    |   movel([0.079939, -1.343105, -2.596200, -0.773084, 1.570796, 1.650735],accel_mss,speed_ms,0,blend_radius_m)
    |   movel([0.079516, -1.343110, -2.596196, -0.773082, 1.570796, 1.650312],accel_mss,speed_ms,0,blend_radius_m)
    |   movel([0.079131, -1.343095, -2.596206, -0.773088, 1.570796, 1.649927],accel_mss,speed_ms,0,blend_radius_m)
    |   movel([0.078857, -1.343061, -2.596229, -0.773099, 1.570796, 1.649653],accel_mss,speed_ms,0,blend_radius_m)
    |   movel([0.077911, -1.342715, -2.596455, -0.773220, 1.570796, 1.648707],accel_mss,speed_ms,0,blend_radius_m)
    |   movel([0.077138, -1.342102, -2.596854, -0.773432, 1.570796, 1.647934],accel_mss,speed_ms,0,blend_radius_m)
    |   movel([0.076602, -1.341277, -2.597392, -0.773720, 1.570796, 1.647398],accel_mss,speed_ms,0,blend_radius_m)
    |   movel([0.076353, -1.340309, -2.598021, -0.774059, 1.570796, 1.647149],accel_mss,speed_ms,0,blend_radius_m)
    |   movel([0.076437, -1.339121, -2.598792, -0.774476, 1.570796, 1.647234],accel_mss,speed_ms,0,blend_radius_m)
    |   movel([0.076894, -1.337754, -2.599676, -0.774958, 1.570796, 1.647690],accel_mss,speed_ms,0,blend_radius_m)
    |   movel([0.077674, -1.336337, -2.600591, -0.775461, 1.570796, 1.648470],accel_mss,speed_ms,0,blend_radius_m)
    |   movel([0.078708, -1.335004, -2.601448, -0.775937, 1.570796, 1.649504],accel_mss,speed_ms,0,blend_radius_m)
    |   movel([0.080811, -1.333153, -2.602635, -0.776601, 1.570796, 1.651607],accel_mss,speed_ms,0,blend_radius_m)
    |   movel([0.083274, -1.331799, -2.603500, -0.777090, 1.570796, 1.654070],accel_mss,speed_ms,0,blend_radius_m)
    |   movel([0.085841, -1.331090, -2.603952, -0.777347, 1.570796, 1.656638],accel_mss,speed_ms,0,blend_radius_m)
    |   movel([0.088231, -1.331107, -2.603941, -0.777341, 1.570796, 1.659028],accel_mss,speed_ms,0,blend_radius_m)
    |   movel([0.089974, -1.331777, -2.603514, -0.777098, 1.570796, 1.660770],accel_mss,speed_ms,0,blend_radius_m)
    |   movel([0.091117, -1.333045, -2.602704, -0.776640, 1.570796, 1.661913],accel_mss,speed_ms,0,blend_radius_m)
    |   movel([0.091521, -1.334728, -2.601626, -0.776036, 1.570796, 1.662317],accel_mss,speed_ms,0,blend_radius_m)
    |   movel([0.091134, -1.336614, -2.600412, -0.775363, 1.570796, 1.661931],accel_mss,speed_ms,0,blend_radius_m)
    |   movel([0.090360, -1.338022, -2.599503, -0.774864, 1.570796, 1.661156],accel_mss,speed_ms,0,blend_radius_m)
    |   movel([0.089237, -1.339332, -2.598656, -0.774402, 1.570796, 1.660033],accel_mss,speed_ms,0,blend_radius_m)
    |   movel([0.087880, -1.340411, -2.597955, -0.774023, 1.570796, 1.658676],accel_mss,speed_ms,0,blend_radius_m)
    |   movel([0.086419, -1.341159, -2.597469, -0.773761, 1.570796, 1.657215],accel_mss,speed_ms,0,blend_radius_m)
    |   movel([0.086085, -1.341294, -2.597381, -0.773714, 1.570796, 1.656881],accel_mss,speed_ms,0,blend_radius_m)
    |   movel([0.085784, -1.341434, -2.597289, -0.773665, 1.570796, 1.656580],accel_mss,speed_ms,0,blend_radius_m)
    |   movel([0.085437, -1.341649, -2.597150, -0.773590, 1.570796, 1.656234],accel_mss,speed_ms,0,blend_radius_m)
    |   movel([0.085272, -1.342062, -2.596880, -0.773446, 1.570796, 1.656068],accel_mss,speed_ms,0,blend_radius_m)
    |   movel([0.085168, -1.342424, -2.596644, -0.773321, 1.570796, 1.655964],accel_mss,speed_ms,0,blend_radius_m)
    |   movel([0.085068, -1.342821, -2.596385, -0.773183, 1.570796, 1.655864],accel_mss,speed_ms,0,blend_radius_m)
    |   movel([0.084872, -1.343546, -2.595911, -0.772931, 1.570796, 1.655669],accel_mss,speed_ms,0,blend_radius_m)
    |   movel([0.084670, -1.343986, -2.595624, -0.772779, 1.570796, 1.655466],accel_mss,speed_ms,0,blend_radius_m)
    |   movel([0.084233, -1.344177, -2.595498, -0.772713, 1.570796, 1.655029],accel_mss,speed_ms,0,blend_radius_m)
    |   movel([0.084159, -1.343630, -2.595857, -0.772903, 1.570796, 1.654955],accel_mss,speed_ms,0,blend_radius_m)
    |   movel([0.084254, -1.342914, -2.596324, -0.773150, 1.570796, 1.655050],accel_mss,speed_ms,0,blend_radius_m)
    |   movel([0.084514, -1.341336, -2.597354, -0.773700, 1.570796, 1.655311],accel_mss,speed_ms,0,blend_radius_m)
    |   movel([0.084702, -1.340274, -2.598044, -0.774071, 1.570796, 1.655498],accel_mss,speed_ms,0,blend_radius_m)
    |   movel([0.084875, -1.339360, -2.598637, -0.774392, 1.570796, 1.655672],accel_mss,speed_ms,0,blend_radius_m)
    |   movel([0.085040, -1.338563, -2.599153, -0.774672, 1.570796, 1.655836],accel_mss,speed_ms,0,blend_radius_m)
    |   movel([0.085311, -1.338276, -2.599339, -0.774774, 1.570796, 1.656107],accel_mss,speed_ms,0,blend_radius_m)
    |   movel([0.085672, -1.338005, -2.599514, -0.774869, 1.570796, 1.656468],accel_mss,speed_ms,0,blend_radius_m)
    |   movel([0.086068, -1.337661, -2.599737, -0.774991, 1.570796, 1.656864],accel_mss,speed_ms,0,blend_radius_m)
    |   movel([0.086444, -1.337219, -2.600022, -0.775148, 1.570796, 1.657240],accel_mss,speed_ms,0,blend_radius_m)
    |   movel([0.086729, -1.336771, -2.600311, -0.775307, 1.570796, 1.657525],accel_mss,speed_ms,0,blend_radius_m)
    |   movel([0.086840, -1.336424, -2.600534, -0.775430, 1.570796, 1.657636],accel_mss,speed_ms,0,blend_radius_m)
    |   movel([0.086756, -1.336163, -2.600703, -0.775523, 1.570796, 1.657553],accel_mss,speed_ms,0,blend_radius_m)
    |   movel([0.086516, -1.335929, -2.600853, -0.775606, 1.570796, 1.657313],accel_mss,speed_ms,0,blend_radius_m)
    |   movel([0.085950, -1.335813, -2.600928, -0.775648, 1.570796, 1.656746],accel_mss,speed_ms,0,blend_radius_m)
    |   movel([0.085372, -1.336061, -2.600768, -0.775559, 1.570796, 1.656169],accel_mss,speed_ms,0,blend_radius_m)
    |   movel([0.084915, -1.336633, -2.600400, -0.775356, 1.570796, 1.655711],accel_mss,speed_ms,0,blend_radius_m)
    |   movel([0.084701, -1.337386, -2.599914, -0.775089, 1.570796, 1.655497],accel_mss,speed_ms,0,blend_radius_m)
    |   movel([0.084629, -1.337702, -2.599710, -0.774977, 1.570796, 1.655425],accel_mss,speed_ms,0,blend_radius_m)
    |   movel([0.084484, -1.338005, -2.599514, -0.774870, 1.570796, 1.655281],accel_mss,speed_ms,0,blend_radius_m)
    |   movel([0.084293, -1.338243, -2.599361, -0.774785, 1.570796, 1.655089],accel_mss,speed_ms,0,blend_radius_m)
    |   movel([0.083838, -1.338404, -2.599256, -0.774729, 1.570796, 1.654634],accel_mss,speed_ms,0,blend_radius_m)
    |   speed_ms = 0.003
    |   movel([0.083838, -1.341807, -2.600812, -0.769770, 1.570796, 1.654634],accel_mss,speed_ms,0,blend_radius_m)
    |   speed_ms = 0.007
    |   movel([0.083575, -1.341756, -2.600845, -0.769788, 1.570796, 1.654371],accel_mss,speed_ms,0,blend_radius_m)
    |   movel([0.083364, -1.341641, -2.600920, -0.769828, 1.570796, 1.654160],accel_mss,speed_ms,0,blend_radius_m)
    |   movel([0.083137, -1.341072, -2.601289, -0.770028, 1.570796, 1.653934],accel_mss,speed_ms,0,blend_radius_m)
    |   movel([0.082925, -1.340755, -2.601495, -0.770139, 1.570796, 1.653721],accel_mss,speed_ms,0,blend_radius_m)
    |   movel([0.082638, -1.340551, -2.601627, -0.770210, 1.570796, 1.653434],accel_mss,speed_ms,0,blend_radius_m)
    |   movel([0.082291, -1.340461, -2.601686, -0.770242, 1.570796, 1.653087],accel_mss,speed_ms,0,blend_radius_m)
    |   movel([0.081838, -1.340482, -2.601672, -0.770235, 1.570796, 1.652635],accel_mss,speed_ms,0,blend_radius_m)
    |   movel([0.081455, -1.340581, -2.601608, -0.770200, 1.570796, 1.652252],accel_mss,speed_ms,0,blend_radius_m)
    |   movel([0.081141, -1.340794, -2.601470, -0.770125, 1.570796, 1.651937],accel_mss,speed_ms,0,blend_radius_m)
    |   movel([0.080784, -1.341164, -2.601229, -0.769995, 1.570796, 1.651580],accel_mss,speed_ms,0,blend_radius_m)
    |   movel([0.080489, -1.341559, -2.600973, -0.769857, 1.570796, 1.651285],accel_mss,speed_ms,0,blend_radius_m)
    |   movel([0.080384, -1.341838, -2.600791, -0.769759, 1.570796, 1.651180],accel_mss,speed_ms,0,blend_radius_m)
    |   movel([0.080469, -1.342126, -2.600605, -0.769659, 1.570796, 1.651266],accel_mss,speed_ms,0,blend_radius_m)
    |   movel([0.080802, -1.342368, -2.600447, -0.769574, 1.570796, 1.651598],accel_mss,speed_ms,0,blend_radius_m)
    |   movel([0.081280, -1.342524, -2.600345, -0.769520, 1.570796, 1.652076],accel_mss,speed_ms,0,blend_radius_m)
    |   movel([0.081829, -1.342556, -2.600324, -0.769508, 1.570796, 1.652625],accel_mss,speed_ms,0,blend_radius_m)
    |   movel([0.082528, -1.342582, -2.600308, -0.769500, 1.570796, 1.653324],accel_mss,speed_ms,0,blend_radius_m)
    |   movel([0.082794, -1.342792, -2.600170, -0.769426, 1.570796, 1.653590],accel_mss,speed_ms,0,blend_radius_m)
    |   movel([0.082846, -1.343313, -2.599831, -0.769245, 1.570796, 1.653642],accel_mss,speed_ms,0,blend_radius_m)
    |   movel([0.082677, -1.345239, -2.598572, -0.768578, 1.570796, 1.653473],accel_mss,speed_ms,0,blend_radius_m)
    |   movel([0.082499, -1.346941, -2.597455, -0.767993, 1.570796, 1.653295],accel_mss,speed_ms,0,blend_radius_m)
    |   movel([0.082356, -1.347693, -2.596960, -0.767736, 1.570796, 1.653152],accel_mss,speed_ms,0,blend_radius_m)
    |   movel([0.082163, -1.348091, -2.596698, -0.767600, 1.570796, 1.652960],accel_mss,speed_ms,0,blend_radius_m)
    |   movel([0.081866, -1.348309, -2.596554, -0.767525, 1.570796, 1.652662],accel_mss,speed_ms,0,blend_radius_m)
    |   movel([0.081568, -1.348137, -2.596668, -0.767584, 1.570796, 1.652364],accel_mss,speed_ms,0,blend_radius_m)
    |   movel([0.081509, -1.347824, -2.596874, -0.767691, 1.570796, 1.652305],accel_mss,speed_ms,0,blend_radius_m)
    |   movel([0.081511, -1.347338, -2.597194, -0.767857, 1.570796, 1.652308],accel_mss,speed_ms,0,blend_radius_m)
    |   movel([0.081515, -1.347062, -2.597375, -0.767951, 1.570796, 1.652311],accel_mss,speed_ms,0,blend_radius_m)
    |   movel([0.081498, -1.346808, -2.597542, -0.768038, 1.570796, 1.652294],accel_mss,speed_ms,0,blend_radius_m)
    |   movel([0.081461, -1.346604, -2.597676, -0.768108, 1.570796, 1.652258],accel_mss,speed_ms,0,blend_radius_m)
    |   movel([0.081307, -1.346463, -2.597769, -0.768157, 1.570796, 1.652103],accel_mss,speed_ms,0,blend_radius_m)
    |   movel([0.081039, -1.346444, -2.597782, -0.768163, 1.570796, 1.651836],accel_mss,speed_ms,0,blend_radius_m)
    |   movel([0.080706, -1.346443, -2.597782, -0.768164, 1.570796, 1.651503],accel_mss,speed_ms,0,blend_radius_m)
    |   movel([0.080338, -1.346469, -2.597765, -0.768155, 1.570796, 1.651134],accel_mss,speed_ms,0,blend_radius_m)
    |   movel([0.079939, -1.346496, -2.597748, -0.768146, 1.570796, 1.650735],accel_mss,speed_ms,0,blend_radius_m)
    |   movel([0.079516, -1.346501, -2.597744, -0.768144, 1.570796, 1.650312],accel_mss,speed_ms,0,blend_radius_m)
    |   movel([0.079131, -1.346486, -2.597754, -0.768149, 1.570796, 1.649927],accel_mss,speed_ms,0,blend_radius_m)
    |   movel([0.078857, -1.346452, -2.597776, -0.768161, 1.570796, 1.649653],accel_mss,speed_ms,0,blend_radius_m)
    |   movel([0.077911, -1.346107, -2.598003, -0.768279, 1.570796, 1.648707],accel_mss,speed_ms,0,blend_radius_m)
    |   movel([0.077138, -1.345496, -2.598404, -0.768490, 1.570796, 1.647934],accel_mss,speed_ms,0,blend_radius_m)
    |   movel([0.076602, -1.344673, -2.598942, -0.768774, 1.570796, 1.647398],accel_mss,speed_ms,0,blend_radius_m)
    |   movel([0.076353, -1.343707, -2.599574, -0.769108, 1.570796, 1.647149],accel_mss,speed_ms,0,blend_radius_m)
    |   movel([0.076437, -1.342522, -2.600346, -0.769520, 1.570796, 1.647234],accel_mss,speed_ms,0,blend_radius_m)
    |   movel([0.076894, -1.341159, -2.601233, -0.769997, 1.570796, 1.647690],accel_mss,speed_ms,0,blend_radius_m)
    |   movel([0.077674, -1.339745, -2.602150, -0.770494, 1.570796, 1.648470],accel_mss,speed_ms,0,blend_radius_m)
    |   movel([0.078708, -1.338415, -2.603009, -0.770964, 1.570796, 1.649504],accel_mss,speed_ms,0,blend_radius_m)
    |   movel([0.080811, -1.336569, -2.604199, -0.771621, 1.570796, 1.651607],accel_mss,speed_ms,0,blend_radius_m)
    |   movel([0.083274, -1.335218, -2.605067, -0.772104, 1.570796, 1.654070],accel_mss,speed_ms,0,blend_radius_m)
    |   movel([0.085841, -1.334511, -2.605520, -0.772358, 1.570796, 1.656638],accel_mss,speed_ms,0,blend_radius_m)
    |   movel([0.088231, -1.334527, -2.605509, -0.772352, 1.570796, 1.659028],accel_mss,speed_ms,0,blend_radius_m)
    |   movel([0.089974, -1.335197, -2.605081, -0.772112, 1.570796, 1.660770],accel_mss,speed_ms,0,blend_radius_m)
    |   movel([0.091117, -1.336461, -2.604269, -0.771659, 1.570796, 1.661913],accel_mss,speed_ms,0,blend_radius_m)
    |   movel([0.091521, -1.338140, -2.603187, -0.771062, 1.570796, 1.662317],accel_mss,speed_ms,0,blend_radius_m)
    |   movel([0.091134, -1.340021, -2.601971, -0.770397, 1.570796, 1.661931],accel_mss,speed_ms,0,blend_radius_m)
    |   movel([0.090360, -1.341426, -2.601060, -0.769904, 1.570796, 1.661156],accel_mss,speed_ms,0,blend_radius_m)
    |   movel([0.089237, -1.342732, -2.600210, -0.769447, 1.570796, 1.660033],accel_mss,speed_ms,0,blend_radius_m)
    |   movel([0.087880, -1.343808, -2.599508, -0.769073, 1.570796, 1.658676],accel_mss,speed_ms,0,blend_radius_m)
    |   movel([0.086419, -1.344555, -2.599020, -0.768814, 1.570796, 1.657215],accel_mss,speed_ms,0,blend_radius_m)
    |   movel([0.086085, -1.344690, -2.598932, -0.768768, 1.570796, 1.656881],accel_mss,speed_ms,0,blend_radius_m)
    |   movel([0.085784, -1.344830, -2.598840, -0.768719, 1.570796, 1.656580],accel_mss,speed_ms,0,blend_radius_m)
    |   movel([0.085437, -1.345043, -2.598700, -0.768646, 1.570796, 1.656234],accel_mss,speed_ms,0,blend_radius_m)
    |   movel([0.085272, -1.345456, -2.598430, -0.768503, 1.570796, 1.656068],accel_mss,speed_ms,0,blend_radius_m)
    |   movel([0.085168, -1.345817, -2.598193, -0.768379, 1.570796, 1.655964],accel_mss,speed_ms,0,blend_radius_m)
    |   movel([0.085068, -1.346213, -2.597933, -0.768243, 1.570796, 1.655864],accel_mss,speed_ms,0,blend_radius_m)
    |   movel([0.084872, -1.346936, -2.597458, -0.767995, 1.570796, 1.655669],accel_mss,speed_ms,0,blend_radius_m)
    |   movel([0.084670, -1.347375, -2.597170, -0.767844, 1.570796, 1.655466],accel_mss,speed_ms,0,blend_radius_m)
    |   movel([0.084233, -1.347565, -2.597044, -0.767779, 1.570796, 1.655029],accel_mss,speed_ms,0,blend_radius_m)
    |   movel([0.084159, -1.347019, -2.597404, -0.767966, 1.570796, 1.654955],accel_mss,speed_ms,0,blend_radius_m)
    |   movel([0.084254, -1.346306, -2.597872, -0.768211, 1.570796, 1.655050],accel_mss,speed_ms,0,blend_radius_m)
    |   movel([0.084514, -1.344731, -2.598904, -0.768754, 1.570796, 1.655311],accel_mss,speed_ms,0,blend_radius_m)
    |   movel([0.084702, -1.343673, -2.599596, -0.769120, 1.570796, 1.655498],accel_mss,speed_ms,0,blend_radius_m)
    |   movel([0.084875, -1.342761, -2.600191, -0.769437, 1.570796, 1.655672],accel_mss,speed_ms,0,blend_radius_m)
    |   movel([0.085040, -1.341966, -2.600709, -0.769715, 1.570796, 1.655836],accel_mss,speed_ms,0,blend_radius_m)
    |   movel([0.085311, -1.341679, -2.600895, -0.769815, 1.570796, 1.656107],accel_mss,speed_ms,0,blend_radius_m)
    |   movel([0.085672, -1.341409, -2.601070, -0.769909, 1.570796, 1.656468],accel_mss,speed_ms,0,blend_radius_m)
    |   movel([0.086068, -1.341066, -2.601294, -0.770030, 1.570796, 1.656864],accel_mss,speed_ms,0,blend_radius_m)
    |   movel([0.086444, -1.340624, -2.601580, -0.770185, 1.570796, 1.657240],accel_mss,speed_ms,0,blend_radius_m)
    |   movel([0.086729, -1.340178, -2.601869, -0.770342, 1.570796, 1.657525],accel_mss,speed_ms,0,blend_radius_m)
    |   movel([0.086840, -1.339832, -2.602093, -0.770464, 1.570796, 1.657636],accel_mss,speed_ms,0,blend_radius_m)
    |   movel([0.086756, -1.339572, -2.602262, -0.770555, 1.570796, 1.657553],accel_mss,speed_ms,0,blend_radius_m)
    |   movel([0.086516, -1.339338, -2.602413, -0.770638, 1.570796, 1.657313],accel_mss,speed_ms,0,blend_radius_m)
    |   movel([0.085950, -1.339222, -2.602488, -0.770679, 1.570796, 1.656746],accel_mss,speed_ms,0,blend_radius_m)
    |   movel([0.085372, -1.339470, -2.602328, -0.770591, 1.570796, 1.656169],accel_mss,speed_ms,0,blend_radius_m)
    |   movel([0.084915, -1.340040, -2.601959, -0.770390, 1.570796, 1.655711],accel_mss,speed_ms,0,blend_radius_m)
    |   movel([0.084701, -1.340791, -2.601472, -0.770126, 1.570796, 1.655497],accel_mss,speed_ms,0,blend_radius_m)
    |   movel([0.084629, -1.341106, -2.601267, -0.770016, 1.570796, 1.655425],accel_mss,speed_ms,0,blend_radius_m)
    |   movel([0.084484, -1.341409, -2.601071, -0.769910, 1.570796, 1.655281],accel_mss,speed_ms,0,blend_radius_m)
    |   movel([0.084293, -1.341646, -2.600916, -0.769826, 1.570796, 1.655089],accel_mss,speed_ms,0,blend_radius_m)
    |   movel([0.083838, -1.341807, -2.600812, -0.769770, 1.570796, 1.654634],accel_mss,speed_ms,0,blend_radius_m)
    |   speed_ms = 0.003
    |   movel([0.083838, -1.328347, -2.594539, -0.789503, 1.570796, 1.654634],accel_mss,speed_ms,0,blend_radius_m)
    |   speed_ms = 1.000
    |   movel([0.083838, -1.302622, -2.581603, -0.828165, 1.570796, 1.654634],accel_mss,speed_ms,0,blend_radius_m)
    |   movel([0.083131, -1.309400, -2.577409, -0.825580, 1.570796, 1.653928],accel_mss,speed_ms,0,blend_radius_m)
    |   movel([0.083131, -1.335017, -2.590258, -0.787114, 1.570796, 1.653928],accel_mss,speed_ms,0,blend_radius_m)
    |   speed_ms = 0.003
    |   movel([0.083131, -1.345027, -2.594942, -0.772421, 1.570796, 1.653928],accel_mss,speed_ms,0,blend_radius_m)
    |   speed_ms = 0.007
    |   movel([0.084912, -1.344646, -2.595191, -0.772552, 1.570796, 1.655708],accel_mss,speed_ms,0,blend_radius_m)
    |   movel([0.085226, -1.344667, -2.595177, -0.772544, 1.570796, 1.656023],accel_mss,speed_ms,0,blend_radius_m)
    |   movel([0.085321, -1.344944, -2.594996, -0.772449, 1.570796, 1.656117],accel_mss,speed_ms,0,blend_radius_m)
    |   movel([0.085214, -1.345307, -2.594758, -0.772325, 1.570796, 1.656010],accel_mss,speed_ms,0,blend_radius_m)
    |   movel([0.085158, -1.345566, -2.594588, -0.772236, 1.570796, 1.655955],accel_mss,speed_ms,0,blend_radius_m)
    |   movel([0.085106, -1.345844, -2.594405, -0.772140, 1.570796, 1.655902],accel_mss,speed_ms,0,blend_radius_m)
    |   movel([0.085067, -1.346106, -2.594233, -0.772050, 1.570796, 1.655864],accel_mss,speed_ms,0,blend_radius_m)
    |   movel([0.085015, -1.346429, -2.594020, -0.771940, 1.570796, 1.655812],accel_mss,speed_ms,0,blend_radius_m)
    |   movel([0.084839, -1.346835, -2.593753, -0.771801, 1.570796, 1.655635],accel_mss,speed_ms,0,blend_radius_m)
    |   movel([0.084290, -1.347303, -2.593444, -0.771641, 1.570796, 1.655087],accel_mss,speed_ms,0,blend_radius_m)
    |   movel([0.083746, -1.347575, -2.593265, -0.771549, 1.570796, 1.654542],accel_mss,speed_ms,0,blend_radius_m)
    |   movel([0.083025, -1.347847, -2.593086, -0.771456, 1.570796, 1.653821],accel_mss,speed_ms,0,blend_radius_m)
    |   movel([0.082091, -1.348128, -2.592900, -0.771361, 1.570796, 1.652888],accel_mss,speed_ms,0,blend_radius_m)
    |   movel([0.081241, -1.348334, -2.592764, -0.771291, 1.570796, 1.652037],accel_mss,speed_ms,0,blend_radius_m)
    |   movel([0.080813, -1.348339, -2.592761, -0.771289, 1.570796, 1.651610],accel_mss,speed_ms,0,blend_radius_m)
    |   movel([0.080675, -1.348167, -2.592874, -0.771347, 1.570796, 1.651471],accel_mss,speed_ms,0,blend_radius_m)
    |   movel([0.080768, -1.347825, -2.593100, -0.771464, 1.570796, 1.651564],accel_mss,speed_ms,0,blend_radius_m)
    |   movel([0.080890, -1.347520, -2.593302, -0.771568, 1.570796, 1.651686],accel_mss,speed_ms,0,blend_radius_m)
    |   movel([0.080645, -1.347327, -2.593429, -0.771633, 1.570796, 1.651441],accel_mss,speed_ms,0,blend_radius_m)
    |   movel([0.080619, -1.347111, -2.593571, -0.771707, 1.570796, 1.651416],accel_mss,speed_ms,0,blend_radius_m)
    |   movel([0.080919, -1.346779, -2.593790, -0.771820, 1.570796, 1.651715],accel_mss,speed_ms,0,blend_radius_m)
    |   movel([0.080769, -1.346426, -2.594022, -0.771941, 1.570796, 1.651566],accel_mss,speed_ms,0,blend_radius_m)
    |   movel([0.080640, -1.346238, -2.594146, -0.772005, 1.570796, 1.651436],accel_mss,speed_ms,0,blend_radius_m)
    |   movel([0.080628, -1.346014, -2.594293, -0.772082, 1.570796, 1.651424],accel_mss,speed_ms,0,blend_radius_m)
    |   movel([0.080942, -1.345606, -2.594561, -0.772222, 1.570796, 1.651739],accel_mss,speed_ms,0,blend_radius_m)
    |   movel([0.081368, -1.345424, -2.594681, -0.772284, 1.570796, 1.652164],accel_mss,speed_ms,0,blend_radius_m)
    |   movel([0.083131, -1.345027, -2.594942, -0.772421, 1.570796, 1.653928],accel_mss,speed_ms,0,blend_radius_m)
    |   speed_ms = 0.003
    |   movel([0.083131, -1.348413, -2.596486, -0.767490, 1.570796, 1.653928],accel_mss,speed_ms,0,blend_radius_m)
    |   speed_ms = 0.007
    |   movel([0.084912, -1.348033, -2.596736, -0.767620, 1.570796, 1.655708],accel_mss,speed_ms,0,blend_radius_m)
    |   movel([0.085226, -1.348054, -2.596722, -0.767612, 1.570796, 1.656023],accel_mss,speed_ms,0,blend_radius_m)
    |   movel([0.085321, -1.348330, -2.596541, -0.767518, 1.570796, 1.656117],accel_mss,speed_ms,0,blend_radius_m)
    |   movel([0.085214, -1.348692, -2.596302, -0.767395, 1.570796, 1.656010],accel_mss,speed_ms,0,blend_radius_m)
    |   movel([0.085158, -1.348950, -2.596131, -0.767307, 1.570796, 1.655955],accel_mss,speed_ms,0,blend_radius_m)
    |   movel([0.085106, -1.349228, -2.595948, -0.767213, 1.570796, 1.655902],accel_mss,speed_ms,0,blend_radius_m)
    |   movel([0.085067, -1.349489, -2.595775, -0.767124, 1.570796, 1.655864],accel_mss,speed_ms,0,blend_radius_m)
    |   movel([0.085015, -1.349812, -2.595562, -0.767015, 1.570796, 1.655812],accel_mss,speed_ms,0,blend_radius_m)
    |   movel([0.084839, -1.350216, -2.595294, -0.766878, 1.570796, 1.655635],accel_mss,speed_ms,0,blend_radius_m)
    |   movel([0.084290, -1.350683, -2.594985, -0.766720, 1.570796, 1.655087],accel_mss,speed_ms,0,blend_radius_m)
    |   movel([0.083746, -1.350954, -2.594806, -0.766629, 1.570796, 1.654542],accel_mss,speed_ms,0,blend_radius_m)
    |   movel([0.083025, -1.351226, -2.594626, -0.766538, 1.570796, 1.653821],accel_mss,speed_ms,0,blend_radius_m)
    |   movel([0.082091, -1.351507, -2.594439, -0.766443, 1.570796, 1.652888],accel_mss,speed_ms,0,blend_radius_m)
    |   movel([0.081241, -1.351712, -2.594303, -0.766374, 1.570796, 1.652037],accel_mss,speed_ms,0,blend_radius_m)
    |   movel([0.080813, -1.351716, -2.594300, -0.766373, 1.570796, 1.651610],accel_mss,speed_ms,0,blend_radius_m)
    |   movel([0.080675, -1.351545, -2.594414, -0.766430, 1.570796, 1.651471],accel_mss,speed_ms,0,blend_radius_m)
    |   movel([0.080768, -1.351204, -2.594640, -0.766545, 1.570796, 1.651564],accel_mss,speed_ms,0,blend_radius_m)
    |   movel([0.080890, -1.350900, -2.594842, -0.766647, 1.570796, 1.651686],accel_mss,speed_ms,0,blend_radius_m)
    |   movel([0.080645, -1.350707, -2.594969, -0.766712, 1.570796, 1.651441],accel_mss,speed_ms,0,blend_radius_m)
    |   movel([0.080619, -1.350492, -2.595112, -0.766785, 1.570796, 1.651416],accel_mss,speed_ms,0,blend_radius_m)
    |   movel([0.080919, -1.350160, -2.595332, -0.766897, 1.570796, 1.651715],accel_mss,speed_ms,0,blend_radius_m)
    |   movel([0.080769, -1.349809, -2.595564, -0.767016, 1.570796, 1.651566],accel_mss,speed_ms,0,blend_radius_m)
    |   movel([0.080640, -1.349621, -2.595688, -0.767080, 1.570796, 1.651436],accel_mss,speed_ms,0,blend_radius_m)
    |   movel([0.080628, -1.349397, -2.595836, -0.767155, 1.570796, 1.651424],accel_mss,speed_ms,0,blend_radius_m)
    |   movel([0.080942, -1.348990, -2.596105, -0.767294, 1.570796, 1.651739],accel_mss,speed_ms,0,blend_radius_m)
    |   movel([0.081368, -1.348809, -2.596225, -0.767355, 1.570796, 1.652164],accel_mss,speed_ms,0,blend_radius_m)
    |   movel([0.083131, -1.348413, -2.596486, -0.767490, 1.570796, 1.653928],accel_mss,speed_ms,0,blend_radius_m)
    |   speed_ms = 0.003
    |   movel([0.083131, -1.335017, -2.590258, -0.787114, 1.570796, 1.653928],accel_mss,speed_ms,0,blend_radius_m)
    |   speed_ms = 1.000
    |   movel([0.083131, -1.309400, -2.577409, -0.825580, 1.570796, 1.653928],accel_mss,speed_ms,0,blend_radius_m)
    |   movel([0.082638, -1.312886, -2.575230, -0.824273, 1.570796, 1.653435],accel_mss,speed_ms,0,blend_radius_m)
    |   movel([0.082638, -1.338446, -2.588033, -0.785910, 1.570796, 1.653435],accel_mss,speed_ms,0,blend_radius_m)
    |   speed_ms = 0.003
    |   movel([0.082638, -1.348431, -2.592700, -0.771258, 1.570796, 1.653435],accel_mss,speed_ms,0,blend_radius_m)
    |   speed_ms = 0.007
    |   movel([0.083010, -1.348325, -2.592770, -0.771294, 1.570796, 1.653806],accel_mss,speed_ms,0,blend_radius_m)
    |   movel([0.083255, -1.348397, -2.592722, -0.771269, 1.570796, 1.654051],accel_mss,speed_ms,0,blend_radius_m)
    |   movel([0.083272, -1.348613, -2.592580, -0.771196, 1.570796, 1.654068],accel_mss,speed_ms,0,blend_radius_m)
    |   movel([0.082991, -1.348882, -2.592402, -0.771105, 1.570796, 1.653788],accel_mss,speed_ms,0,blend_radius_m)
    |   movel([0.082561, -1.349059, -2.592285, -0.771045, 1.570796, 1.653357],accel_mss,speed_ms,0,blend_radius_m)
    |   movel([0.082329, -1.349028, -2.592305, -0.771056, 1.570796, 1.653125],accel_mss,speed_ms,0,blend_radius_m)
    |   movel([0.082337, -1.348676, -2.592538, -0.771175, 1.570796, 1.653134],accel_mss,speed_ms,0,blend_radius_m)
    |   movel([0.082638, -1.348431, -2.592700, -0.771258, 1.570796, 1.653435],accel_mss,speed_ms,0,blend_radius_m)
    |   speed_ms = 0.003
    |   movel([0.082638, -1.351808, -2.594239, -0.766342, 1.570796, 1.653435],accel_mss,speed_ms,0,blend_radius_m)
    |   speed_ms = 0.007
    |   movel([0.083010, -1.351702, -2.594309, -0.766377, 1.570796, 1.653806],accel_mss,speed_ms,0,blend_radius_m)
    |   movel([0.083255, -1.351775, -2.594261, -0.766353, 1.570796, 1.654051],accel_mss,speed_ms,0,blend_radius_m)
    |   movel([0.083272, -1.351990, -2.594118, -0.766281, 1.570796, 1.654068],accel_mss,speed_ms,0,blend_radius_m)
    |   movel([0.082991, -1.352258, -2.593940, -0.766191, 1.570796, 1.653788],accel_mss,speed_ms,0,blend_radius_m)
    |   movel([0.082561, -1.352435, -2.593823, -0.766132, 1.570796, 1.653357],accel_mss,speed_ms,0,blend_radius_m)
    |   movel([0.082329, -1.352404, -2.593843, -0.766142, 1.570796, 1.653125],accel_mss,speed_ms,0,blend_radius_m)
    |   movel([0.082337, -1.352052, -2.594077, -0.766260, 1.570796, 1.653134],accel_mss,speed_ms,0,blend_radius_m)
    |   movel([0.082638, -1.351808, -2.594239, -0.766342, 1.570796, 1.653435],accel_mss,speed_ms,0,blend_radius_m)
    |   speed_ms = 0.003
    |   movel([0.082638, -1.338446, -2.588033, -0.785910, 1.570796, 1.653435],accel_mss,speed_ms,0,blend_radius_m)
    |   speed_ms = 1.000
    |   movel([0.082638, -1.312886, -2.575230, -0.824273, 1.570796, 1.653435],accel_mss,speed_ms,0,blend_radius_m)
    |   movel([0.075847, -1.319560, -2.571014, -0.821815, 1.570796, 1.646643],accel_mss,speed_ms,0,blend_radius_m)
    |   movel([0.075847, -1.345010, -2.583731, -0.783648, 1.570796, 1.646643],accel_mss,speed_ms,0,blend_radius_m)
    |   speed_ms = 0.003
    |   movel([0.075847, -1.354947, -2.588365, -0.769077, 1.570796, 1.646643],accel_mss,speed_ms,0,blend_radius_m)
    |   speed_ms = 0.007
    |   movel([0.076210, -1.355243, -2.588167, -0.768979, 1.570796, 1.647006],accel_mss,speed_ms,0,blend_radius_m)
    |   movel([0.076357, -1.355481, -2.588008, -0.768901, 1.570796, 1.647154],accel_mss,speed_ms,0,blend_radius_m)
    |   movel([0.076398, -1.355704, -2.587858, -0.768827, 1.570796, 1.647194],accel_mss,speed_ms,0,blend_radius_m)
    |   movel([0.076337, -1.355959, -2.587687, -0.768743, 1.570796, 1.647134],accel_mss,speed_ms,0,blend_radius_m)
    |   movel([0.076172, -1.356294, -2.587462, -0.768633, 1.570796, 1.646969],accel_mss,speed_ms,0,blend_radius_m)
    |   movel([0.075752, -1.356855, -2.587085, -0.768449, 1.570796, 1.646548],accel_mss,speed_ms,0,blend_radius_m)
    |   movel([0.075239, -1.357270, -2.586806, -0.768313, 1.570796, 1.646035],accel_mss,speed_ms,0,blend_radius_m)
    |   movel([0.074675, -1.357502, -2.586649, -0.768238, 1.570796, 1.645471],accel_mss,speed_ms,0,blend_radius_m)
    |   movel([0.074114, -1.357533, -2.586628, -0.768227, 1.570796, 1.644910],accel_mss,speed_ms,0,blend_radius_m)
    |   movel([0.073609, -1.357253, -2.586817, -0.768319, 1.570796, 1.644405],accel_mss,speed_ms,0,blend_radius_m)
    |   movel([0.073464, -1.356659, -2.587216, -0.768513, 1.570796, 1.644260],accel_mss,speed_ms,0,blend_radius_m)
    |   movel([0.073721, -1.355938, -2.587701, -0.768750, 1.570796, 1.644518],accel_mss,speed_ms,0,blend_radius_m)
    |   movel([0.074305, -1.355315, -2.588118, -0.768955, 1.570796, 1.645101],accel_mss,speed_ms,0,blend_radius_m)
    |   movel([0.074876, -1.354985, -2.588340, -0.769064, 1.570796, 1.645673],accel_mss,speed_ms,0,blend_radius_m)
    |   movel([0.075398, -1.354858, -2.588425, -0.769106, 1.570796, 1.646194],accel_mss,speed_ms,0,blend_radius_m)
    |   movel([0.075847, -1.354947, -2.588365, -0.769077, 1.570796, 1.646643],accel_mss,speed_ms,0,blend_radius_m)
    |   speed_ms = 0.003
    |   movel([0.075847, -1.358308, -2.589893, -0.764188, 1.570796, 1.646643],accel_mss,speed_ms,0,blend_radius_m)
    |   speed_ms = 0.007
    |   movel([0.076210, -1.358603, -2.589694, -0.764092, 1.570796, 1.647006],accel_mss,speed_ms,0,blend_radius_m)
    |   movel([0.076357, -1.358840, -2.589535, -0.764014, 1.570796, 1.647154],accel_mss,speed_ms,0,blend_radius_m)
    |   movel([0.076398, -1.359063, -2.589385, -0.763942, 1.570796, 1.647194],accel_mss,speed_ms,0,blend_radius_m)
    |   movel([0.076337, -1.359317, -2.589213, -0.763859, 1.570796, 1.647134],accel_mss,speed_ms,0,blend_radius_m)
    |   movel([0.076172, -1.359651, -2.588988, -0.763751, 1.570796, 1.646969],accel_mss,speed_ms,0,blend_radius_m)
    |   movel([0.075752, -1.360211, -2.588610, -0.763569, 1.570796, 1.646548],accel_mss,speed_ms,0,blend_radius_m)
    |   movel([0.075239, -1.360624, -2.588330, -0.763435, 1.570796, 1.646035],accel_mss,speed_ms,0,blend_radius_m)
    |   movel([0.074675, -1.360856, -2.588173, -0.763360, 1.570796, 1.645471],accel_mss,speed_ms,0,blend_radius_m)
    |   movel([0.074114, -1.360887, -2.588152, -0.763350, 1.570796, 1.644910],accel_mss,speed_ms,0,blend_radius_m)
    |   movel([0.073609, -1.360608, -2.588341, -0.763440, 1.570796, 1.644405],accel_mss,speed_ms,0,blend_radius_m)
    |   movel([0.073464, -1.360015, -2.588742, -0.763632, 1.570796, 1.644260],accel_mss,speed_ms,0,blend_radius_m)
    |   movel([0.073721, -1.359296, -2.589227, -0.763866, 1.570796, 1.644518],accel_mss,speed_ms,0,blend_radius_m)
    |   movel([0.074305, -1.358675, -2.589646, -0.764068, 1.570796, 1.645101],accel_mss,speed_ms,0,blend_radius_m)
    |   movel([0.074876, -1.358345, -2.589868, -0.764176, 1.570796, 1.645673],accel_mss,speed_ms,0,blend_radius_m)
    |   movel([0.075398, -1.358219, -2.589953, -0.764217, 1.570796, 1.646194],accel_mss,speed_ms,0,blend_radius_m)
    |   movel([0.075847, -1.358308, -2.589893, -0.764188, 1.570796, 1.646643],accel_mss,speed_ms,0,blend_radius_m)
    |   speed_ms = 0.003
    |   movel([0.075847, -1.345010, -2.583731, -0.783648, 1.570796, 1.646643],accel_mss,speed_ms,0,blend_radius_m)
    |   speed_ms = 1.000
    |   movel([0.075847, -1.319560, -2.571014, -0.821815, 1.570796, 1.646643],accel_mss,speed_ms,0,blend_radius_m)
    |   movel([0.078635, -1.323961, -2.568202, -0.820226, 1.570796, 1.649431],accel_mss,speed_ms,0,blend_radius_m)
    |   movel([0.078635, -1.349337, -2.580862, -0.782189, 1.570796, 1.649431],accel_mss,speed_ms,0,blend_radius_m)
    |   speed_ms = 0.003
    |   movel([0.078635, -1.359242, -2.585475, -0.767671, 1.570796, 1.649431],accel_mss,speed_ms,0,blend_radius_m)
    |   speed_ms = 0.007
    |   movel([0.079474, -1.359723, -2.585151, -0.767516, 1.570796, 1.650271],accel_mss,speed_ms,0,blend_radius_m)
    |   movel([0.080172, -1.360238, -2.584802, -0.767349, 1.570796, 1.650969],accel_mss,speed_ms,0,blend_radius_m)
    |   movel([0.080222, -1.360455, -2.584655, -0.767279, 1.570796, 1.651018],accel_mss,speed_ms,0,blend_radius_m)
    |   movel([0.079954, -1.360655, -2.584519, -0.767215, 1.570796, 1.650750],accel_mss,speed_ms,0,blend_radius_m)
    |   movel([0.079275, -1.360021, -2.584949, -0.767419, 1.570796, 1.650071],accel_mss,speed_ms,0,blend_radius_m)
    |   movel([0.078610, -1.359377, -2.585384, -0.767628, 1.570796, 1.649406],accel_mss,speed_ms,0,blend_radius_m)
    |   speed_ms = 0.003
    |   movel([0.078635, -1.362592, -2.586996, -0.762801, 1.570796, 1.649431],accel_mss,speed_ms,0,blend_radius_m)
    |   speed_ms = 0.007
    |   movel([0.079474, -1.363071, -2.586671, -0.762648, 1.570796, 1.650271],accel_mss,speed_ms,0,blend_radius_m)
    |   movel([0.080172, -1.363585, -2.586321, -0.762483, 1.570796, 1.650969],accel_mss,speed_ms,0,blend_radius_m)
    |   movel([0.080222, -1.363801, -2.586174, -0.762414, 1.570796, 1.651018],accel_mss,speed_ms,0,blend_radius_m)
    |   movel([0.079954, -1.364001, -2.586038, -0.762350, 1.570796, 1.650750],accel_mss,speed_ms,0,blend_radius_m)
    |   movel([0.079275, -1.363368, -2.586468, -0.762552, 1.570796, 1.650071],accel_mss,speed_ms,0,blend_radius_m)
    |   movel([0.078610, -1.362726, -2.586905, -0.762758, 1.570796, 1.649406],accel_mss,speed_ms,0,blend_radius_m)
    |   speed_ms = 0.003
    |   movel([0.078635, -1.349337, -2.580862, -0.782189, 1.570796, 1.649431],accel_mss,speed_ms,0,blend_radius_m)
    |   speed_ms = 1.000
    |   movel([0.078635, -1.323961, -2.568202, -0.820226, 1.570796, 1.649431],accel_mss,speed_ms,0,blend_radius_m)
    |   movel([0.084889, -1.331749, -2.563164, -0.817476, 1.570796, 1.655685],accel_mss,speed_ms,0,blend_radius_m)
    |   movel([0.084889, -1.356993, -2.575725, -0.779672, 1.570796, 1.655685],accel_mss,speed_ms,0,blend_radius_m)
    |   speed_ms = 0.003
    |   movel([0.084889, -1.366841, -2.580300, -0.765248, 1.570796, 1.655685],accel_mss,speed_ms,0,blend_radius_m)
    |   speed_ms = 0.007
    |   movel([0.085264, -1.366718, -2.580384, -0.765287, 1.570796, 1.656061],accel_mss,speed_ms,0,blend_radius_m)
    |   movel([0.085429, -1.367001, -2.580190, -0.765198, 1.570796, 1.656225],accel_mss,speed_ms,0,blend_radius_m)
    |   movel([0.085290, -1.367254, -2.580016, -0.765119, 1.570796, 1.656086],accel_mss,speed_ms,0,blend_radius_m)
    |   movel([0.085006, -1.367407, -2.579911, -0.765071, 1.570796, 1.655802],accel_mss,speed_ms,0,blend_radius_m)
    |   movel([0.084700, -1.367358, -2.579945, -0.765087, 1.570796, 1.655496],accel_mss,speed_ms,0,blend_radius_m)
    |   movel([0.084687, -1.367140, -2.580094, -0.765155, 1.570796, 1.655483],accel_mss,speed_ms,0,blend_radius_m)
    |   movel([0.084889, -1.366841, -2.580300, -0.765248, 1.570796, 1.655685],accel_mss,speed_ms,0,blend_radius_m)
    |   speed_ms = 0.003
    |   movel([0.084889, -1.370170, -2.581808, -0.760411, 1.570796, 1.655685],accel_mss,speed_ms,0,blend_radius_m)
    |   speed_ms = 0.007
    |   movel([0.085264, -1.370048, -2.581893, -0.760449, 1.570796, 1.656061],accel_mss,speed_ms,0,blend_radius_m)
    |   movel([0.085429, -1.370330, -2.581698, -0.760361, 1.570796, 1.656225],accel_mss,speed_ms,0,blend_radius_m)
    |   movel([0.085290, -1.370582, -2.581524, -0.760283, 1.570796, 1.656086],accel_mss,speed_ms,0,blend_radius_m)
    |   movel([0.085006, -1.370735, -2.581418, -0.760236, 1.570796, 1.655802],accel_mss,speed_ms,0,blend_radius_m)
    |   movel([0.084700, -1.370686, -2.581452, -0.760251, 1.570796, 1.655496],accel_mss,speed_ms,0,blend_radius_m)
    |   movel([0.084687, -1.370469, -2.581602, -0.760318, 1.570796, 1.655483],accel_mss,speed_ms,0,blend_radius_m)
    |   movel([0.084889, -1.370170, -2.581808, -0.760411, 1.570796, 1.655685],accel_mss,speed_ms,0,blend_radius_m)
    |   speed_ms = 0.003
    |   movel([0.084889, -1.356993, -2.575725, -0.779672, 1.570796, 1.655685],accel_mss,speed_ms,0,blend_radius_m)
    |   speed_ms = 1.000
    |   movel([0.084889, -1.331749, -2.563164, -0.817476, 1.570796, 1.655685],accel_mss,speed_ms,0,blend_radius_m)
    |   movel([0.086824, -1.329871, -2.564386, -0.818131, 1.570796, 1.657620],accel_mss,speed_ms,0,blend_radius_m)
    |   movel([0.086824, -1.355147, -2.576970, -0.780271, 1.570796, 1.657620],accel_mss,speed_ms,0,blend_radius_m)
    |   speed_ms = 0.003
    |   movel([0.086824, -1.365009, -2.581555, -0.765825, 1.570796, 1.657620],accel_mss,speed_ms,0,blend_radius_m)
    |   speed_ms = 0.007
    |   movel([0.087168, -1.365279, -2.581370, -0.765740, 1.570796, 1.657964],accel_mss,speed_ms,0,blend_radius_m)
    |   movel([0.087391, -1.365516, -2.581208, -0.765665, 1.570796, 1.658187],accel_mss,speed_ms,0,blend_radius_m)
    |   movel([0.087551, -1.365788, -2.581021, -0.765579, 1.570796, 1.658347],accel_mss,speed_ms,0,blend_radius_m)
    |   movel([0.087693, -1.366165, -2.580764, -0.765461, 1.570796, 1.658489],accel_mss,speed_ms,0,blend_radius_m)
    |   movel([0.087762, -1.366699, -2.580397, -0.765293, 1.570796, 1.658558],accel_mss,speed_ms,0,blend_radius_m)
    |   movel([0.087686, -1.367444, -2.579885, -0.765060, 1.570796, 1.658482],accel_mss,speed_ms,0,blend_radius_m)
    |   movel([0.087505, -1.368211, -2.579358, -0.764820, 1.570796, 1.658301],accel_mss,speed_ms,0,blend_radius_m)
    |   movel([0.087241, -1.368817, -2.578940, -0.764632, 1.570796, 1.658038],accel_mss,speed_ms,0,blend_radius_m)
    |   movel([0.086827, -1.369458, -2.578498, -0.764433, 1.570796, 1.657623],accel_mss,speed_ms,0,blend_radius_m)
    |   movel([0.086336, -1.370058, -2.578084, -0.764247, 1.570796, 1.657133],accel_mss,speed_ms,0,blend_radius_m)
    |   movel([0.085769, -1.370615, -2.577699, -0.764075, 1.570796, 1.656565],accel_mss,speed_ms,0,blend_radius_m)
    |   movel([0.085120, -1.371138, -2.577337, -0.763914, 1.570796, 1.655916],accel_mss,speed_ms,0,blend_radius_m)
    |   movel([0.084603, -1.371499, -2.577086, -0.763803, 1.570796, 1.655399],accel_mss,speed_ms,0,blend_radius_m)
    |   movel([0.084238, -1.371707, -2.576942, -0.763740, 1.570796, 1.655035],accel_mss,speed_ms,0,blend_radius_m)
    |   movel([0.083834, -1.371872, -2.576828, -0.763689, 1.570796, 1.654631],accel_mss,speed_ms,0,blend_radius_m)
    |   movel([0.083145, -1.372087, -2.576679, -0.763623, 1.570796, 1.653941],accel_mss,speed_ms,0,blend_radius_m)
    |   movel([0.082486, -1.372273, -2.576550, -0.763566, 1.570796, 1.653282],accel_mss,speed_ms,0,blend_radius_m)
    |   movel([0.082081, -1.372352, -2.576495, -0.763542, 1.570796, 1.652877],accel_mss,speed_ms,0,blend_radius_m)
    |   movel([0.081735, -1.372366, -2.576485, -0.763538, 1.570796, 1.652532],accel_mss,speed_ms,0,blend_radius_m)
    |   movel([0.081304, -1.372326, -2.576513, -0.763550, 1.570796, 1.652101],accel_mss,speed_ms,0,blend_radius_m)
    |   movel([0.080718, -1.372180, -2.576614, -0.763595, 1.570796, 1.651515],accel_mss,speed_ms,0,blend_radius_m)
    |   movel([0.080185, -1.371922, -2.576793, -0.763674, 1.570796, 1.650981],accel_mss,speed_ms,0,blend_radius_m)
    |   movel([0.079747, -1.371571, -2.577037, -0.763781, 1.570796, 1.650544],accel_mss,speed_ms,0,blend_radius_m)
    |   movel([0.079442, -1.371152, -2.577327, -0.763910, 1.570796, 1.650238],accel_mss,speed_ms,0,blend_radius_m)
    |   movel([0.079335, -1.370890, -2.577508, -0.763991, 1.570796, 1.650132],accel_mss,speed_ms,0,blend_radius_m)
    |   movel([0.079280, -1.370612, -2.577701, -0.764076, 1.570796, 1.650076],accel_mss,speed_ms,0,blend_radius_m)
    |   movel([0.079271, -1.370257, -2.577947, -0.764186, 1.570796, 1.650067],accel_mss,speed_ms,0,blend_radius_m)
    |   movel([0.079306, -1.369743, -2.578301, -0.764344, 1.570796, 1.650102],accel_mss,speed_ms,0,blend_radius_m)
    |   movel([0.079370, -1.369178, -2.578691, -0.764520, 1.570796, 1.650167],accel_mss,speed_ms,0,blend_radius_m)
    |   movel([0.079452, -1.368805, -2.578949, -0.764635, 1.570796, 1.650248],accel_mss,speed_ms,0,blend_radius_m)
    |   movel([0.079585, -1.368463, -2.579184, -0.764742, 1.570796, 1.650381],accel_mss,speed_ms,0,blend_radius_m)
    |   movel([0.079810, -1.368029, -2.579483, -0.764877, 1.570796, 1.650606],accel_mss,speed_ms,0,blend_radius_m)
    |   movel([0.080321, -1.367272, -2.580004, -0.765113, 1.570796, 1.651117],accel_mss,speed_ms,0,blend_radius_m)
    |   movel([0.080995, -1.366513, -2.580524, -0.765351, 1.570796, 1.651792],accel_mss,speed_ms,0,blend_radius_m)
    |   movel([0.081741, -1.365848, -2.580980, -0.765560, 1.570796, 1.652537],accel_mss,speed_ms,0,blend_radius_m)
    |   movel([0.082465, -1.365369, -2.581309, -0.765711, 1.570796, 1.653262],accel_mss,speed_ms,0,blend_radius_m)
    |   movel([0.083702, -1.364840, -2.581671, -0.765879, 1.570796, 1.654499],accel_mss,speed_ms,0,blend_radius_m)
    |   movel([0.084908, -1.364595, -2.581838, -0.765956, 1.570796, 1.655704],accel_mss,speed_ms,0,blend_radius_m)
    |   movel([0.085979, -1.364652, -2.581799, -0.765938, 1.570796, 1.656775],accel_mss,speed_ms,0,blend_radius_m)
    |   movel([0.086824, -1.365009, -2.581555, -0.765825, 1.570796, 1.657620],accel_mss,speed_ms,0,blend_radius_m)
    |   speed_ms = 0.003
    |   movel([0.086824, -1.368344, -2.583066, -0.760979, 1.570796, 1.657620],accel_mss,speed_ms,0,blend_radius_m)
    |   speed_ms = 0.007
    |   movel([0.087168, -1.368612, -2.582881, -0.760896, 1.570796, 1.657964],accel_mss,speed_ms,0,blend_radius_m)
    |   movel([0.087391, -1.368849, -2.582719, -0.760822, 1.570796, 1.658187],accel_mss,speed_ms,0,blend_radius_m)
    |   movel([0.087551, -1.369121, -2.582531, -0.760737, 1.570796, 1.658347],accel_mss,speed_ms,0,blend_radius_m)
    |   movel([0.087693, -1.369496, -2.582273, -0.760620, 1.570796, 1.658489],accel_mss,speed_ms,0,blend_radius_m)
    |   movel([0.087762, -1.370029, -2.581906, -0.760455, 1.570796, 1.658558],accel_mss,speed_ms,0,blend_radius_m)
    |   movel([0.087686, -1.370772, -2.581393, -0.760224, 1.570796, 1.658482],accel_mss,speed_ms,0,blend_radius_m)
    |   movel([0.087505, -1.371537, -2.580864, -0.759988, 1.570796, 1.658301],accel_mss,speed_ms,0,blend_radius_m)
    |   movel([0.087241, -1.372141, -2.580445, -0.759802, 1.570796, 1.658038],accel_mss,speed_ms,0,blend_radius_m)
    |   movel([0.086827, -1.372781, -2.580002, -0.759606, 1.570796, 1.657623],accel_mss,speed_ms,0,blend_radius_m)
    |   movel([0.086336, -1.373379, -2.579587, -0.759423, 1.570796, 1.657133],accel_mss,speed_ms,0,blend_radius_m)
    |   movel([0.085769, -1.373934, -2.579201, -0.759254, 1.570796, 1.656565],accel_mss,speed_ms,0,blend_radius_m)
    |   movel([0.085120, -1.374456, -2.578838, -0.759095, 1.570796, 1.655916],accel_mss,speed_ms,0,blend_radius_m)
    |   movel([0.084603, -1.374816, -2.578587, -0.758986, 1.570796, 1.655399],accel_mss,speed_ms,0,blend_radius_m)
    |   movel([0.084238, -1.375023, -2.578443, -0.758923, 1.570796, 1.655035],accel_mss,speed_ms,0,blend_radius_m)
    |   movel([0.083834, -1.375188, -2.578328, -0.758873, 1.570796, 1.654631],accel_mss,speed_ms,0,blend_radius_m)
    |   movel([0.083145, -1.375403, -2.578178, -0.758808, 1.570796, 1.653941],accel_mss,speed_ms,0,blend_radius_m)
    |   movel([0.082486, -1.375588, -2.578049, -0.758752, 1.570796, 1.653282],accel_mss,speed_ms,0,blend_radius_m)
    |   movel([0.082081, -1.375667, -2.577994, -0.758728, 1.570796, 1.652877],accel_mss,speed_ms,0,blend_radius_m)
    |   movel([0.081735, -1.375681, -2.577984, -0.758724, 1.570796, 1.652532],accel_mss,speed_ms,0,blend_radius_m)
    |   movel([0.081304, -1.375641, -2.578012, -0.758736, 1.570796, 1.652101],accel_mss,speed_ms,0,blend_radius_m)
    |   movel([0.080718, -1.375495, -2.578114, -0.758780, 1.570796, 1.651515],accel_mss,speed_ms,0,blend_radius_m)
    |   movel([0.080185, -1.375238, -2.578293, -0.758858, 1.570796, 1.650981],accel_mss,speed_ms,0,blend_radius_m)
    |   movel([0.079747, -1.374887, -2.578537, -0.758964, 1.570796, 1.650544],accel_mss,speed_ms,0,blend_radius_m)
    |   movel([0.079442, -1.374470, -2.578828, -0.759091, 1.570796, 1.650238],accel_mss,speed_ms,0,blend_radius_m)
    |   movel([0.079335, -1.374209, -2.579010, -0.759170, 1.570796, 1.650132],accel_mss,speed_ms,0,blend_radius_m)
    |   movel([0.079280, -1.373932, -2.579203, -0.759255, 1.570796, 1.650076],accel_mss,speed_ms,0,blend_radius_m)
    |   movel([0.079271, -1.373577, -2.579449, -0.759363, 1.570796, 1.650067],accel_mss,speed_ms,0,blend_radius_m)
    |   movel([0.079306, -1.373065, -2.579805, -0.759519, 1.570796, 1.650102],accel_mss,speed_ms,0,blend_radius_m)
    |   movel([0.079370, -1.372501, -2.580196, -0.759692, 1.570796, 1.650167],accel_mss,speed_ms,0,blend_radius_m)
    |   movel([0.079452, -1.372129, -2.580454, -0.759806, 1.570796, 1.650248],accel_mss,speed_ms,0,blend_radius_m)
    |   movel([0.079585, -1.371788, -2.580690, -0.759911, 1.570796, 1.650381],accel_mss,speed_ms,0,blend_radius_m)
    |   movel([0.079810, -1.371355, -2.580990, -0.760044, 1.570796, 1.650606],accel_mss,speed_ms,0,blend_radius_m)
    |   movel([0.080321, -1.370600, -2.581511, -0.760278, 1.570796, 1.651117],accel_mss,speed_ms,0,blend_radius_m)
    |   movel([0.080995, -1.369844, -2.582033, -0.760512, 1.570796, 1.651792],accel_mss,speed_ms,0,blend_radius_m)
    |   movel([0.081741, -1.369180, -2.582490, -0.760718, 1.570796, 1.652537],accel_mss,speed_ms,0,blend_radius_m)
    |   movel([0.082465, -1.368702, -2.582819, -0.760867, 1.570796, 1.653262],accel_mss,speed_ms,0,blend_radius_m)
    |   movel([0.083702, -1.368175, -2.583182, -0.761032, 1.570796, 1.654499],accel_mss,speed_ms,0,blend_radius_m)
    |   movel([0.084908, -1.367930, -2.583350, -0.761109, 1.570796, 1.655704],accel_mss,speed_ms,0,blend_radius_m)
    |   movel([0.085979, -1.367988, -2.583311, -0.761091, 1.570796, 1.656775],accel_mss,speed_ms,0,blend_radius_m)
    |   movel([0.086824, -1.368344, -2.583066, -0.760979, 1.570796, 1.657620],accel_mss,speed_ms,0,blend_radius_m)
    |   speed_ms = 0.003
    |   movel([0.086824, -1.355147, -2.576970, -0.780271, 1.570796, 1.657620],accel_mss,speed_ms,0,blend_radius_m)
    |   speed_ms = 1.000
    |   movel([0.086824, -1.329871, -2.564386, -0.818131, 1.570796, 1.657620],accel_mss,speed_ms,0,blend_radius_m)
    |   movel([0.094772, -1.328855, -2.565045, -0.818488, 1.570796, 1.665569],accel_mss,speed_ms,0,blend_radius_m)
    |   movel([0.094772, -1.354149, -2.577643, -0.780598, 1.570796, 1.665569],accel_mss,speed_ms,0,blend_radius_m)
    |   speed_ms = 0.003
    |   movel([0.094772, -1.364018, -2.582232, -0.766139, 1.570796, 1.665569],accel_mss,speed_ms,0,blend_radius_m)
    |   speed_ms = 0.007
    |   movel([0.094995, -1.363677, -2.582465, -0.766248, 1.570796, 1.665791],accel_mss,speed_ms,0,blend_radius_m)
    |   movel([0.095323, -1.363701, -2.582448, -0.766240, 1.570796, 1.666120],accel_mss,speed_ms,0,blend_radius_m)
    |   movel([0.095419, -1.363975, -2.582261, -0.766153, 1.570796, 1.666215],accel_mss,speed_ms,0,blend_radius_m)
    |   movel([0.095125, -1.364292, -2.582045, -0.766052, 1.570796, 1.665921],accel_mss,speed_ms,0,blend_radius_m)
    |   movel([0.094811, -1.364341, -2.582011, -0.766037, 1.570796, 1.665607],accel_mss,speed_ms,0,blend_radius_m)
    |   movel([0.094772, -1.364018, -2.582232, -0.766139, 1.570796, 1.665569],accel_mss,speed_ms,0,blend_radius_m)
    |   speed_ms = 0.003
    |   movel([0.094772, -1.367355, -2.583745, -0.761289, 1.570796, 1.665569],accel_mss,speed_ms,0,blend_radius_m)
    |   speed_ms = 0.007
    |   movel([0.094995, -1.367014, -2.583978, -0.761396, 1.570796, 1.665791],accel_mss,speed_ms,0,blend_radius_m)
    |   movel([0.095323, -1.367038, -2.583962, -0.761389, 1.570796, 1.666120],accel_mss,speed_ms,0,blend_radius_m)
    |   movel([0.095419, -1.367312, -2.583774, -0.761303, 1.570796, 1.666215],accel_mss,speed_ms,0,blend_radius_m)
    |   movel([0.095125, -1.367628, -2.583557, -0.761203, 1.570796, 1.665921],accel_mss,speed_ms,0,blend_radius_m)
    |   movel([0.094811, -1.367677, -2.583524, -0.761188, 1.570796, 1.665607],accel_mss,speed_ms,0,blend_radius_m)
    |   movel([0.094772, -1.367355, -2.583745, -0.761289, 1.570796, 1.665569],accel_mss,speed_ms,0,blend_radius_m)
    |   speed_ms = 0.003
    |   movel([0.094772, -1.354149, -2.577643, -0.780598, 1.570796, 1.665569],accel_mss,speed_ms,0,blend_radius_m)
    |   speed_ms = 1.000
    |   movel([0.094772, -1.328855, -2.565045, -0.818488, 1.570796, 1.665569],accel_mss,speed_ms,0,blend_radius_m)
    |   movel([0.093044, -1.328349, -2.565373, -0.818667, 1.570796, 1.663841],accel_mss,speed_ms,0,blend_radius_m)
    |   movel([0.093044, -1.353651, -2.577977, -0.780761, 1.570796, 1.663841],accel_mss,speed_ms,0,blend_radius_m)
    |   speed_ms = 0.003
    |   movel([0.093044, -1.363524, -2.582569, -0.766296, 1.570796, 1.663841],accel_mss,speed_ms,0,blend_radius_m)
    |   speed_ms = 0.007
    |   movel([0.093644, -1.362822, -2.583047, -0.766520, 1.570796, 1.664441],accel_mss,speed_ms,0,blend_radius_m)
    |   movel([0.094331, -1.362169, -2.583491, -0.766728, 1.570796, 1.665128],accel_mss,speed_ms,0,blend_radius_m)
    |   movel([0.095046, -1.361633, -2.583856, -0.766900, 1.570796, 1.665842],accel_mss,speed_ms,0,blend_radius_m)
    |   movel([0.096773, -1.360824, -2.584405, -0.767160, 1.570796, 1.667569],accel_mss,speed_ms,0,blend_radius_m)
    |   movel([0.098461, -1.360629, -2.584537, -0.767223, 1.570796, 1.669258],accel_mss,speed_ms,0,blend_radius_m)
    |   movel([0.099813, -1.361083, -2.584229, -0.767077, 1.570796, 1.670609],accel_mss,speed_ms,0,blend_radius_m)
    |   movel([0.100589, -1.362108, -2.583533, -0.766748, 1.570796, 1.671385],accel_mss,speed_ms,0,blend_radius_m)
    |   movel([0.100651, -1.362593, -2.583203, -0.766593, 1.570796, 1.671448],accel_mss,speed_ms,0,blend_radius_m)
    |   movel([0.100652, -1.362928, -2.582975, -0.766486, 1.570796, 1.671448],accel_mss,speed_ms,0,blend_radius_m)
    |   movel([0.100628, -1.363261, -2.582748, -0.766380, 1.570796, 1.671424],accel_mss,speed_ms,0,blend_radius_m)
    |   movel([0.100362, -1.364362, -2.581997, -0.766030, 1.570796, 1.671159],accel_mss,speed_ms,0,blend_radius_m)
    |   movel([0.099808, -1.365429, -2.581267, -0.765692, 1.570796, 1.670604],accel_mss,speed_ms,0,blend_radius_m)
    |   movel([0.098981, -1.366422, -2.580587, -0.765380, 1.570796, 1.669777],accel_mss,speed_ms,0,blend_radius_m)
    |   movel([0.097911, -1.367310, -2.579977, -0.765101, 1.570796, 1.668707],accel_mss,speed_ms,0,blend_radius_m)
    |   movel([0.097420, -1.367637, -2.579752, -0.764999, 1.570796, 1.668216],accel_mss,speed_ms,0,blend_radius_m)
    |   movel([0.097050, -1.367840, -2.579613, -0.764936, 1.570796, 1.667847],accel_mss,speed_ms,0,blend_radius_m)
    |   movel([0.096644, -1.368002, -2.579502, -0.764885, 1.570796, 1.667440],accel_mss,speed_ms,0,blend_radius_m)
    |   movel([0.096013, -1.368199, -2.579366, -0.764824, 1.570796, 1.666809],accel_mss,speed_ms,0,blend_radius_m)
    |   movel([0.095377, -1.368373, -2.579247, -0.764770, 1.570796, 1.666173],accel_mss,speed_ms,0,blend_radius_m)
    |   movel([0.094976, -1.368446, -2.579196, -0.764747, 1.570796, 1.665772],accel_mss,speed_ms,0,blend_radius_m)
    |   movel([0.094614, -1.368453, -2.579191, -0.764745, 1.570796, 1.665410],accel_mss,speed_ms,0,blend_radius_m)
    |   movel([0.094128, -1.368401, -2.579227, -0.764761, 1.570796, 1.664925],accel_mss,speed_ms,0,blend_radius_m)
    |   movel([0.093507, -1.368260, -2.579324, -0.764805, 1.570796, 1.664303],accel_mss,speed_ms,0,blend_radius_m)
    |   movel([0.093023, -1.368028, -2.579484, -0.764877, 1.570796, 1.663819],accel_mss,speed_ms,0,blend_radius_m)
    |   movel([0.092642, -1.367684, -2.579721, -0.764985, 1.570796, 1.663438],accel_mss,speed_ms,0,blend_radius_m)
    |   movel([0.092324, -1.367203, -2.580051, -0.765135, 1.570796, 1.663120],accel_mss,speed_ms,0,blend_radius_m)
    |   movel([0.092145, -1.366594, -2.580469, -0.765326, 1.570796, 1.662941],accel_mss,speed_ms,0,blend_radius_m)
    |   movel([0.092139, -1.365795, -2.581017, -0.765577, 1.570796, 1.662936],accel_mss,speed_ms,0,blend_radius_m)
    |   movel([0.092293, -1.364952, -2.581594, -0.765843, 1.570796, 1.663090],accel_mss,speed_ms,0,blend_radius_m)
    |   movel([0.092597, -1.364210, -2.582101, -0.766078, 1.570796, 1.663394],accel_mss,speed_ms,0,blend_radius_m)
    |   movel([0.093044, -1.363524, -2.582569, -0.766296, 1.570796, 1.663841],accel_mss,speed_ms,0,blend_radius_m)
    |   speed_ms = 0.003
    |   movel([0.093044, -1.366862, -2.584083, -0.761444, 1.570796, 1.663841],accel_mss,speed_ms,0,blend_radius_m)
    |   speed_ms = 0.007
    |   movel([0.093644, -1.366162, -2.584562, -0.761665, 1.570796, 1.664441],accel_mss,speed_ms,0,blend_radius_m)
    |   movel([0.094331, -1.365511, -2.585007, -0.761871, 1.570796, 1.665128],accel_mss,speed_ms,0,blend_radius_m)
    |   movel([0.095046, -1.364976, -2.585373, -0.762040, 1.570796, 1.665842],accel_mss,speed_ms,0,blend_radius_m)
    |   movel([0.096773, -1.364169, -2.585923, -0.762297, 1.570796, 1.667569],accel_mss,speed_ms,0,blend_radius_m)
    |   movel([0.098461, -1.363974, -2.586056, -0.762359, 1.570796, 1.669258],accel_mss,speed_ms,0,blend_radius_m)
    |   movel([0.099813, -1.364427, -2.585747, -0.762215, 1.570796, 1.670609],accel_mss,speed_ms,0,blend_radius_m)
    |   movel([0.100589, -1.365450, -2.585049, -0.761890, 1.570796, 1.671385],accel_mss,speed_ms,0,blend_radius_m)
    |   movel([0.100651, -1.365933, -2.584718, -0.761737, 1.570796, 1.671448],accel_mss,speed_ms,0,blend_radius_m)
    |   movel([0.100652, -1.366267, -2.584490, -0.761632, 1.570796, 1.671448],accel_mss,speed_ms,0,blend_radius_m)
    |   movel([0.100628, -1.366600, -2.584262, -0.761527, 1.570796, 1.671424],accel_mss,speed_ms,0,blend_radius_m)
    |   movel([0.100362, -1.367698, -2.583509, -0.761181, 1.570796, 1.671159],accel_mss,speed_ms,0,blend_radius_m)
    |   movel([0.099808, -1.368763, -2.582778, -0.760849, 1.570796, 1.670604],accel_mss,speed_ms,0,blend_radius_m)
    |   movel([0.098981, -1.369752, -2.582096, -0.760540, 1.570796, 1.669777],accel_mss,speed_ms,0,blend_radius_m)
    |   movel([0.097911, -1.370638, -2.581485, -0.760266, 1.570796, 1.668707],accel_mss,speed_ms,0,blend_radius_m)
    |   movel([0.097420, -1.370965, -2.581259, -0.760165, 1.570796, 1.668216],accel_mss,speed_ms,0,blend_radius_m)
    |   movel([0.097050, -1.371167, -2.581120, -0.760103, 1.570796, 1.667847],accel_mss,speed_ms,0,blend_radius_m)
    |   movel([0.096644, -1.371328, -2.581008, -0.760053, 1.570796, 1.667440],accel_mss,speed_ms,0,blend_radius_m)
    |   movel([0.096013, -1.371525, -2.580872, -0.759992, 1.570796, 1.666809],accel_mss,speed_ms,0,blend_radius_m)
    |   movel([0.095377, -1.371698, -2.580752, -0.759939, 1.570796, 1.666173],accel_mss,speed_ms,0,blend_radius_m)
    |   movel([0.094976, -1.371771, -2.580701, -0.759916, 1.570796, 1.665772],accel_mss,speed_ms,0,blend_radius_m)
    |   movel([0.094614, -1.371778, -2.580697, -0.759914, 1.570796, 1.665410],accel_mss,speed_ms,0,blend_radius_m)
    |   movel([0.094128, -1.371726, -2.580733, -0.759930, 1.570796, 1.664925],accel_mss,speed_ms,0,blend_radius_m)
    |   movel([0.093507, -1.371585, -2.580830, -0.759973, 1.570796, 1.664303],accel_mss,speed_ms,0,blend_radius_m)
    |   movel([0.093023, -1.371354, -2.580990, -0.760045, 1.570796, 1.663819],accel_mss,speed_ms,0,blend_radius_m)
    |   movel([0.092642, -1.371011, -2.581228, -0.760151, 1.570796, 1.663438],accel_mss,speed_ms,0,blend_radius_m)
    |   movel([0.092324, -1.370532, -2.581559, -0.760299, 1.570796, 1.663120],accel_mss,speed_ms,0,blend_radius_m)
    |   movel([0.092145, -1.369924, -2.581978, -0.760487, 1.570796, 1.662941],accel_mss,speed_ms,0,blend_radius_m)
    |   movel([0.092139, -1.369127, -2.582527, -0.760735, 1.570796, 1.662936],accel_mss,speed_ms,0,blend_radius_m)
    |   movel([0.092293, -1.368287, -2.583105, -0.760997, 1.570796, 1.663090],accel_mss,speed_ms,0,blend_radius_m)
    |   movel([0.092597, -1.367547, -2.583613, -0.761229, 1.570796, 1.663394],accel_mss,speed_ms,0,blend_radius_m)
    |   movel([0.093044, -1.366862, -2.584083, -0.761444, 1.570796, 1.663841],accel_mss,speed_ms,0,blend_radius_m)
    |   speed_ms = 0.003
    |   movel([0.093044, -1.353651, -2.577977, -0.780761, 1.570796, 1.663841],accel_mss,speed_ms,0,blend_radius_m)
    |   speed_ms = 1.000
    |   movel([0.093044, -1.328349, -2.565373, -0.818667, 1.570796, 1.663841],accel_mss,speed_ms,0,blend_radius_m)
    |   movel([0.093095, -1.337880, -2.559143, -0.815367, 1.570796, 1.663891],accel_mss,speed_ms,0,blend_radius_m)
    |   movel([0.093095, -1.363017, -2.571624, -0.777747, 1.570796, 1.663891],accel_mss,speed_ms,0,blend_radius_m)
    |   speed_ms = 0.003
    |   movel([0.093095, -1.372820, -2.576170, -0.763399, 1.570796, 1.663891],accel_mss,speed_ms,0,blend_radius_m)
    |   speed_ms = 0.007
    |   movel([0.095667, -1.371889, -2.576816, -0.763684, 1.570796, 1.666464],accel_mss,speed_ms,0,blend_radius_m)
    |   movel([0.097439, -1.371146, -2.577331, -0.763912, 1.570796, 1.668235],accel_mss,speed_ms,0,blend_radius_m)
    |   movel([0.099151, -1.370361, -2.577874, -0.764154, 1.570796, 1.669947],accel_mss,speed_ms,0,blend_radius_m)
    |   movel([0.100738, -1.369566, -2.578424, -0.764399, 1.570796, 1.671535],accel_mss,speed_ms,0,blend_radius_m)
    |   movel([0.102129, -1.368796, -2.578955, -0.764638, 1.570796, 1.672925],accel_mss,speed_ms,0,blend_radius_m)
    |   movel([0.103079, -1.368244, -2.579335, -0.764810, 1.570796, 1.673875],accel_mss,speed_ms,0,blend_radius_m)
    |   movel([0.103407, -1.368085, -2.579445, -0.764859, 1.570796, 1.674203],accel_mss,speed_ms,0,blend_radius_m)
    |   movel([0.103782, -1.368141, -2.579406, -0.764842, 1.570796, 1.674579],accel_mss,speed_ms,0,blend_radius_m)
    |   movel([0.103972, -1.368477, -2.579175, -0.764737, 1.570796, 1.674769],accel_mss,speed_ms,0,blend_radius_m)
    |   movel([0.104047, -1.369268, -2.578630, -0.764492, 1.570796, 1.674843],accel_mss,speed_ms,0,blend_radius_m)
    |   movel([0.104025, -1.370097, -2.578057, -0.764235, 1.570796, 1.674822],accel_mss,speed_ms,0,blend_radius_m)
    |   movel([0.103868, -1.370632, -2.577687, -0.764070, 1.570796, 1.674664],accel_mss,speed_ms,0,blend_radius_m)
    |   movel([0.103307, -1.371174, -2.577312, -0.763903, 1.570796, 1.674104],accel_mss,speed_ms,0,blend_radius_m)
    |   movel([0.100371, -1.372580, -2.576336, -0.763472, 1.570796, 1.671167],accel_mss,speed_ms,0,blend_radius_m)
    |   movel([0.097202, -1.373985, -2.575359, -0.763045, 1.570796, 1.667998],accel_mss,speed_ms,0,blend_radius_m)
    |   movel([0.094275, -1.375126, -2.574563, -0.762700, 1.570796, 1.665072],accel_mss,speed_ms,0,blend_radius_m)
    |   movel([0.091963, -1.375881, -2.574036, -0.762472, 1.570796, 1.662759],accel_mss,speed_ms,0,blend_radius_m)
    |   movel([0.088651, -1.376817, -2.573380, -0.762191, 1.570796, 1.659447],accel_mss,speed_ms,0,blend_radius_m)
    |   movel([0.085300, -1.377694, -2.572766, -0.761930, 1.570796, 1.656096],accel_mss,speed_ms,0,blend_radius_m)
    |   movel([0.082794, -1.378255, -2.572372, -0.761763, 1.570796, 1.653590],accel_mss,speed_ms,0,blend_radius_m)
    |   movel([0.080908, -1.378590, -2.572136, -0.761663, 1.570796, 1.651704],accel_mss,speed_ms,0,blend_radius_m)
    |   movel([0.078698, -1.378923, -2.571902, -0.761564, 1.570796, 1.649495],accel_mss,speed_ms,0,blend_radius_m)
    |   movel([0.076615, -1.379200, -2.571707, -0.761482, 1.570796, 1.647412],accel_mss,speed_ms,0,blend_radius_m)
    |   movel([0.075933, -1.379208, -2.571701, -0.761480, 1.570796, 1.646730],accel_mss,speed_ms,0,blend_radius_m)
    |   movel([0.075687, -1.379042, -2.571818, -0.761529, 1.570796, 1.646483],accel_mss,speed_ms,0,blend_radius_m)
    |   movel([0.075673, -1.378811, -2.571981, -0.761597, 1.570796, 1.646469],accel_mss,speed_ms,0,blend_radius_m)
    |   movel([0.075722, -1.378205, -2.572406, -0.761777, 1.570796, 1.646518],accel_mss,speed_ms,0,blend_radius_m)
    |   movel([0.075826, -1.377463, -2.572928, -0.761998, 1.570796, 1.646623],accel_mss,speed_ms,0,blend_radius_m)
    |   movel([0.075986, -1.376875, -2.573340, -0.762174, 1.570796, 1.646783],accel_mss,speed_ms,0,blend_radius_m)
    |   movel([0.076193, -1.376445, -2.573641, -0.762303, 1.570796, 1.646990],accel_mss,speed_ms,0,blend_radius_m)
    |   movel([0.076445, -1.376205, -2.573809, -0.762375, 1.570796, 1.647241],accel_mss,speed_ms,0,blend_radius_m)
    |   movel([0.076934, -1.376110, -2.573875, -0.762403, 1.570796, 1.647730],accel_mss,speed_ms,0,blend_radius_m)
    |   movel([0.077336, -1.376082, -2.573895, -0.762412, 1.570796, 1.648132],accel_mss,speed_ms,0,blend_radius_m)
    |   movel([0.077768, -1.376072, -2.573902, -0.762415, 1.570796, 1.648564],accel_mss,speed_ms,0,blend_radius_m)
    |   movel([0.078966, -1.376038, -2.573926, -0.762425, 1.570796, 1.649762],accel_mss,speed_ms,0,blend_radius_m)
    |   movel([0.080402, -1.375921, -2.574008, -0.762460, 1.570796, 1.651198],accel_mss,speed_ms,0,blend_radius_m)
    |   movel([0.081934, -1.375738, -2.574136, -0.762515, 1.570796, 1.652730],accel_mss,speed_ms,0,blend_radius_m)
    |   movel([0.083427, -1.375504, -2.574300, -0.762586, 1.570796, 1.654223],accel_mss,speed_ms,0,blend_radius_m)
    |   movel([0.085813, -1.374972, -2.574671, -0.762746, 1.570796, 1.656609],accel_mss,speed_ms,0,blend_radius_m)
    |   movel([0.089434, -1.373949, -2.575384, -0.763056, 1.570796, 1.660230],accel_mss,speed_ms,0,blend_radius_m)
    |   movel([0.093095, -1.372820, -2.576170, -0.763399, 1.570796, 1.663891],accel_mss,speed_ms,0,blend_radius_m)
    |   speed_ms = 0.003
    |   movel([0.093095, -1.376133, -2.577668, -0.758587, 1.570796, 1.663891],accel_mss,speed_ms,0,blend_radius_m)
    |   speed_ms = 0.007
    |   movel([0.095667, -1.375205, -2.578316, -0.758868, 1.570796, 1.666464],accel_mss,speed_ms,0,blend_radius_m)
    |   movel([0.097439, -1.374463, -2.578833, -0.759093, 1.570796, 1.668235],accel_mss,speed_ms,0,blend_radius_m)
    |   movel([0.099151, -1.373681, -2.579377, -0.759331, 1.570796, 1.669947],accel_mss,speed_ms,0,blend_radius_m)
    |   movel([0.100738, -1.372888, -2.579927, -0.759573, 1.570796, 1.671535],accel_mss,speed_ms,0,blend_radius_m)
    |   movel([0.102129, -1.372121, -2.580460, -0.759809, 1.570796, 1.672925],accel_mss,speed_ms,0,blend_radius_m)
    |   movel([0.103079, -1.371569, -2.580841, -0.759978, 1.570796, 1.673875],accel_mss,speed_ms,0,blend_radius_m)
    |   movel([0.103407, -1.371411, -2.580951, -0.760027, 1.570796, 1.674203],accel_mss,speed_ms,0,blend_radius_m)
    |   movel([0.103782, -1.371467, -2.580912, -0.760010, 1.570796, 1.674579],accel_mss,speed_ms,0,blend_radius_m)
    |   movel([0.103972, -1.371802, -2.580680, -0.759907, 1.570796, 1.674769],accel_mss,speed_ms,0,blend_radius_m)
    |   movel([0.104047, -1.372591, -2.580134, -0.759665, 1.570796, 1.674843],accel_mss,speed_ms,0,blend_radius_m)
    |   movel([0.104025, -1.373418, -2.579560, -0.759411, 1.570796, 1.674822],accel_mss,speed_ms,0,blend_radius_m)
    |   movel([0.103868, -1.373951, -2.579189, -0.759249, 1.570796, 1.674664],accel_mss,speed_ms,0,blend_radius_m)
    |   movel([0.103307, -1.374492, -2.578813, -0.759084, 1.570796, 1.674104],accel_mss,speed_ms,0,blend_radius_m)
    |   movel([0.100371, -1.375894, -2.577835, -0.758659, 1.570796, 1.671167],accel_mss,speed_ms,0,blend_radius_m)
    |   movel([0.097202, -1.377295, -2.576856, -0.758238, 1.570796, 1.667998],accel_mss,speed_ms,0,blend_radius_m)
    |   movel([0.094275, -1.378433, -2.576058, -0.757898, 1.570796, 1.665072],accel_mss,speed_ms,0,blend_radius_m)
    |   movel([0.091963, -1.379186, -2.575529, -0.757674, 1.570796, 1.662759],accel_mss,speed_ms,0,blend_radius_m)
    |   movel([0.088651, -1.380120, -2.574872, -0.757397, 1.570796, 1.659447],accel_mss,speed_ms,0,blend_radius_m)
    |   movel([0.085300, -1.380994, -2.574256, -0.757139, 1.570796, 1.656096],accel_mss,speed_ms,0,blend_radius_m)
    |   movel([0.082794, -1.381553, -2.573861, -0.756974, 1.570796, 1.653590],accel_mss,speed_ms,0,blend_radius_m)
    |   movel([0.080908, -1.381888, -2.573625, -0.756876, 1.570796, 1.651704],accel_mss,speed_ms,0,blend_radius_m)
    |   movel([0.078698, -1.382220, -2.573390, -0.756779, 1.570796, 1.649495],accel_mss,speed_ms,0,blend_radius_m)
    |   movel([0.076615, -1.382497, -2.573195, -0.756698, 1.570796, 1.647412],accel_mss,speed_ms,0,blend_radius_m)
    |   movel([0.075933, -1.382504, -2.573189, -0.756696, 1.570796, 1.646730],accel_mss,speed_ms,0,blend_radius_m)
    |   movel([0.075687, -1.382338, -2.573307, -0.756744, 1.570796, 1.646483],accel_mss,speed_ms,0,blend_radius_m)
    |   movel([0.075673, -1.382108, -2.573469, -0.756812, 1.570796, 1.646469],accel_mss,speed_ms,0,blend_radius_m)
    |   movel([0.075722, -1.381504, -2.573896, -0.756989, 1.570796, 1.646518],accel_mss,speed_ms,0,blend_radius_m)
    |   movel([0.075826, -1.380764, -2.574419, -0.757207, 1.570796, 1.646623],accel_mss,speed_ms,0,blend_radius_m)
    |   movel([0.075986, -1.380177, -2.574832, -0.757380, 1.570796, 1.646783],accel_mss,speed_ms,0,blend_radius_m)
    |   movel([0.076193, -1.379748, -2.575134, -0.757507, 1.570796, 1.646990],accel_mss,speed_ms,0,blend_radius_m)
    |   movel([0.076445, -1.379509, -2.575302, -0.757578, 1.570796, 1.647241],accel_mss,speed_ms,0,blend_radius_m)
    |   movel([0.076934, -1.379415, -2.575368, -0.757606, 1.570796, 1.647730],accel_mss,speed_ms,0,blend_radius_m)
    |   movel([0.077336, -1.379386, -2.575388, -0.757614, 1.570796, 1.648132],accel_mss,speed_ms,0,blend_radius_m)
    |   movel([0.077768, -1.379376, -2.575395, -0.757617, 1.570796, 1.648564],accel_mss,speed_ms,0,blend_radius_m)
    |   movel([0.078966, -1.379343, -2.575419, -0.757627, 1.570796, 1.649762],accel_mss,speed_ms,0,blend_radius_m)
    |   movel([0.080402, -1.379226, -2.575501, -0.757662, 1.570796, 1.651198],accel_mss,speed_ms,0,blend_radius_m)
    |   movel([0.081934, -1.379044, -2.575629, -0.757716, 1.570796, 1.652730],accel_mss,speed_ms,0,blend_radius_m)
    |   movel([0.083427, -1.378810, -2.575794, -0.757786, 1.570796, 1.654223],accel_mss,speed_ms,0,blend_radius_m)
    |   movel([0.085813, -1.378280, -2.576166, -0.757944, 1.570796, 1.656609],accel_mss,speed_ms,0,blend_radius_m)
    |   movel([0.089434, -1.377259, -2.576881, -0.758249, 1.570796, 1.660230],accel_mss,speed_ms,0,blend_radius_m)
    |   movel([0.093095, -1.376133, -2.577668, -0.758587, 1.570796, 1.663891],accel_mss,speed_ms,0,blend_radius_m)
    |   speed_ms = 0.003
    |   movel([0.093095, -1.363017, -2.571624, -0.777747, 1.570796, 1.663891],accel_mss,speed_ms,0,blend_radius_m)
    |   speed_ms = 1.000
    |   movel([0.093095, -1.337880, -2.559143, -0.815367, 1.570796, 1.663891],accel_mss,speed_ms,0,blend_radius_m)
    |   movel([0.094637, -1.340831, -2.557189, -0.814369, 1.570796, 1.665433],accel_mss,speed_ms,0,blend_radius_m)
    |   movel([0.094637, -1.365917, -2.569633, -0.776839, 1.570796, 1.665433],accel_mss,speed_ms,0,blend_radius_m)
    |   speed_ms = 0.003
    |   movel([0.094637, -1.375697, -2.574164, -0.762527, 1.570796, 1.665433],accel_mss,speed_ms,0,blend_radius_m)
    |   speed_ms = 0.007
    |   movel([0.094653, -1.376219, -2.573799, -0.762371, 1.570796, 1.665449],accel_mss,speed_ms,0,blend_radius_m)
    |   movel([0.094666, -1.376607, -2.573528, -0.762254, 1.570796, 1.665463],accel_mss,speed_ms,0,blend_radius_m)
    |   movel([0.094670, -1.376842, -2.573363, -0.762184, 1.570796, 1.665466],accel_mss,speed_ms,0,blend_radius_m)
    |   movel([0.094469, -1.377074, -2.573201, -0.762115, 1.570796, 1.665265],accel_mss,speed_ms,0,blend_radius_m)
    |   movel([0.094064, -1.377312, -2.573034, -0.762044, 1.570796, 1.664860],accel_mss,speed_ms,0,blend_radius_m)
    |   movel([0.090980, -1.378254, -2.572372, -0.761763, 1.570796, 1.661777],accel_mss,speed_ms,0,blend_radius_m)
    |   movel([0.088110, -1.379102, -2.571776, -0.761511, 1.570796, 1.658906],accel_mss,speed_ms,0,blend_radius_m)
    |   movel([0.086332, -1.379547, -2.571462, -0.761379, 1.570796, 1.657129],accel_mss,speed_ms,0,blend_radius_m)
    |   movel([0.085492, -1.379705, -2.571351, -0.761333, 1.570796, 1.656288],accel_mss,speed_ms,0,blend_radius_m)
    |   movel([0.085165, -1.379666, -2.571378, -0.761344, 1.570796, 1.655961],accel_mss,speed_ms,0,blend_radius_m)
    |   movel([0.085064, -1.379455, -2.571527, -0.761407, 1.570796, 1.655861],accel_mss,speed_ms,0,blend_radius_m)
    |   movel([0.085171, -1.378948, -2.571884, -0.761557, 1.570796, 1.655967],accel_mss,speed_ms,0,blend_radius_m)
    |   movel([0.085340, -1.378391, -2.572276, -0.761722, 1.570796, 1.656137],accel_mss,speed_ms,0,blend_radius_m)
    |   movel([0.089986, -1.377037, -2.573226, -0.762125, 1.570796, 1.660782],accel_mss,speed_ms,0,blend_radius_m)
    |   movel([0.094637, -1.375697, -2.574164, -0.762527, 1.570796, 1.665433],accel_mss,speed_ms,0,blend_radius_m)
    |   speed_ms = 0.003
    |   movel([0.094637, -1.379003, -2.575658, -0.757728, 1.570796, 1.665433],accel_mss,speed_ms,0,blend_radius_m)
    |   speed_ms = 0.007
    |   movel([0.094653, -1.379524, -2.575292, -0.757573, 1.570796, 1.665449],accel_mss,speed_ms,0,blend_radius_m)
    |   movel([0.094666, -1.379910, -2.575020, -0.757459, 1.570796, 1.665463],accel_mss,speed_ms,0,blend_radius_m)
    |   movel([0.094670, -1.380144, -2.574855, -0.757390, 1.570796, 1.665466],accel_mss,speed_ms,0,blend_radius_m)
    |   movel([0.094469, -1.380376, -2.574692, -0.757321, 1.570796, 1.665265],accel_mss,speed_ms,0,blend_radius_m)
    |   movel([0.094064, -1.380613, -2.574525, -0.757251, 1.570796, 1.664860],accel_mss,speed_ms,0,blend_radius_m)
    |   movel([0.090980, -1.381553, -2.573862, -0.756974, 1.570796, 1.661777],accel_mss,speed_ms,0,blend_radius_m)
    |   movel([0.088110, -1.382398, -2.573264, -0.756727, 1.570796, 1.658906],accel_mss,speed_ms,0,blend_radius_m)
    |   movel([0.086332, -1.382843, -2.572950, -0.756597, 1.570796, 1.657129],accel_mss,speed_ms,0,blend_radius_m)
    |   movel([0.085492, -1.382999, -2.572838, -0.756551, 1.570796, 1.656288],accel_mss,speed_ms,0,blend_radius_m)
    |   movel([0.085165, -1.382961, -2.572866, -0.756562, 1.570796, 1.655961],accel_mss,speed_ms,0,blend_radius_m)
    |   movel([0.085064, -1.382750, -2.573015, -0.756624, 1.570796, 1.655861],accel_mss,speed_ms,0,blend_radius_m)
    |   movel([0.085171, -1.382245, -2.573372, -0.756771, 1.570796, 1.655967],accel_mss,speed_ms,0,blend_radius_m)
    |   movel([0.085340, -1.381689, -2.573765, -0.756934, 1.570796, 1.656137],accel_mss,speed_ms,0,blend_radius_m)
    |   movel([0.089986, -1.380339, -2.574718, -0.757332, 1.570796, 1.660782],accel_mss,speed_ms,0,blend_radius_m)
    |   movel([0.094637, -1.379003, -2.575658, -0.757728, 1.570796, 1.665433],accel_mss,speed_ms,0,blend_radius_m)
    |   speed_ms = 0.003
    |   movel([0.094637, -1.365917, -2.569633, -0.776839, 1.570796, 1.665433],accel_mss,speed_ms,0,blend_radius_m)
    |   speed_ms = 1.000
    |   movel([0.094637, -1.340831, -2.557189, -0.814369, 1.570796, 1.665433],accel_mss,speed_ms,0,blend_radius_m)
    |   movel([0.094776, -1.347374, -2.552816, -0.812199, 1.570796, 1.665572],accel_mss,speed_ms,0,blend_radius_m)
    |   movel([0.094776, -1.372344, -2.565176, -0.774868, 1.570796, 1.665572],accel_mss,speed_ms,0,blend_radius_m)
    |   speed_ms = 0.003
    |   movel([0.094776, -1.382075, -2.569677, -0.760637, 1.570796, 1.665572],accel_mss,speed_ms,0,blend_radius_m)
    |   speed_ms = 0.007
    |   movel([0.096440, -1.381462, -2.570110, -0.760816, 1.570796, 1.667237],accel_mss,speed_ms,0,blend_radius_m)
    |   movel([0.096911, -1.381238, -2.570269, -0.760882, 1.570796, 1.667707],accel_mss,speed_ms,0,blend_radius_m)
    |   movel([0.097314, -1.381204, -2.570293, -0.760892, 1.570796, 1.668110],accel_mss,speed_ms,0,blend_radius_m)
    |   movel([0.097422, -1.381359, -2.570183, -0.760846, 1.570796, 1.668218],accel_mss,speed_ms,0,blend_radius_m)
    |   movel([0.097435, -1.381607, -2.570008, -0.760774, 1.570796, 1.668231],accel_mss,speed_ms,0,blend_radius_m)
    |   movel([0.097301, -1.382148, -2.569625, -0.760616, 1.570796, 1.668098],accel_mss,speed_ms,0,blend_radius_m)
    |   movel([0.097178, -1.382558, -2.569334, -0.760496, 1.570796, 1.667974],accel_mss,speed_ms,0,blend_radius_m)
    |   movel([0.097039, -1.382977, -2.569037, -0.760375, 1.570796, 1.667835],accel_mss,speed_ms,0,blend_radius_m)
    |   movel([0.096697, -1.383916, -2.568371, -0.760103, 1.570796, 1.667493],accel_mss,speed_ms,0,blend_radius_m)
    |   movel([0.096287, -1.384945, -2.567638, -0.759806, 1.570796, 1.667084],accel_mss,speed_ms,0,blend_radius_m)
    |   movel([0.095880, -1.385915, -2.566946, -0.759527, 1.570796, 1.666677],accel_mss,speed_ms,0,blend_radius_m)
    |   movel([0.095733, -1.386137, -2.566788, -0.759464, 1.570796, 1.666529],accel_mss,speed_ms,0,blend_radius_m)
    |   movel([0.095575, -1.385999, -2.566887, -0.759503, 1.570796, 1.666371],accel_mss,speed_ms,0,blend_radius_m)
    |   movel([0.095465, -1.385691, -2.567106, -0.759592, 1.570796, 1.666261],accel_mss,speed_ms,0,blend_radius_m)
    |   movel([0.095361, -1.385540, -2.567214, -0.759635, 1.570796, 1.666157],accel_mss,speed_ms,0,blend_radius_m)
    |   movel([0.095087, -1.385336, -2.567360, -0.759694, 1.570796, 1.665884],accel_mss,speed_ms,0,blend_radius_m)
    |   movel([0.094829, -1.385186, -2.567466, -0.759737, 1.570796, 1.665625],accel_mss,speed_ms,0,blend_radius_m)
    |   movel([0.094690, -1.385009, -2.567592, -0.759787, 1.570796, 1.665486],accel_mss,speed_ms,0,blend_radius_m)
    |   movel([0.094486, -1.384711, -2.567805, -0.759873, 1.570796, 1.665282],accel_mss,speed_ms,0,blend_radius_m)
    |   movel([0.093913, -1.384330, -2.568076, -0.759983, 1.570796, 1.664709],accel_mss,speed_ms,0,blend_radius_m)
    |   movel([0.093257, -1.383995, -2.568314, -0.760080, 1.570796, 1.664053],accel_mss,speed_ms,0,blend_radius_m)
    |   movel([0.092692, -1.383834, -2.568428, -0.760126, 1.570796, 1.663488],accel_mss,speed_ms,0,blend_radius_m)
    |   movel([0.092049, -1.383769, -2.568475, -0.760145, 1.570796, 1.662845],accel_mss,speed_ms,0,blend_radius_m)
    |   movel([0.091353, -1.383774, -2.568471, -0.760144, 1.570796, 1.662149],accel_mss,speed_ms,0,blend_radius_m)
    |   movel([0.090674, -1.383839, -2.568425, -0.760125, 1.570796, 1.661470],accel_mss,speed_ms,0,blend_radius_m)
    |   movel([0.090083, -1.383966, -2.568335, -0.760088, 1.570796, 1.660879],accel_mss,speed_ms,0,blend_radius_m)
    |   movel([0.089683, -1.384047, -2.568277, -0.760065, 1.570796, 1.660479],accel_mss,speed_ms,0,blend_radius_m)
    |   movel([0.089967, -1.383735, -2.568499, -0.760155, 1.570796, 1.660763],accel_mss,speed_ms,0,blend_radius_m)
    |   movel([0.090498, -1.383539, -2.568638, -0.760212, 1.570796, 1.661294],accel_mss,speed_ms,0,blend_radius_m)
    |   movel([0.091427, -1.383232, -2.568856, -0.760301, 1.570796, 1.662224],accel_mss,speed_ms,0,blend_radius_m)
    |   movel([0.093010, -1.382702, -2.569233, -0.760455, 1.570796, 1.663806],accel_mss,speed_ms,0,blend_radius_m)
    |   movel([0.094776, -1.382075, -2.569677, -0.760637, 1.570796, 1.665572],accel_mss,speed_ms,0,blend_radius_m)
    |   speed_ms = 0.003
    |   movel([0.094776, -1.385364, -2.571160, -0.755866, 1.570796, 1.665572],accel_mss,speed_ms,0,blend_radius_m)
    |   speed_ms = 0.007
    |   movel([0.096440, -1.384753, -2.571594, -0.756042, 1.570796, 1.667237],accel_mss,speed_ms,0,blend_radius_m)
    |   movel([0.096911, -1.384529, -2.571754, -0.756107, 1.570796, 1.667707],accel_mss,speed_ms,0,blend_radius_m)
    |   movel([0.097314, -1.384495, -2.571778, -0.756117, 1.570796, 1.668110],accel_mss,speed_ms,0,blend_radius_m)
    |   movel([0.097422, -1.384650, -2.571667, -0.756072, 1.570796, 1.668218],accel_mss,speed_ms,0,blend_radius_m)
    |   movel([0.097435, -1.384896, -2.571492, -0.756001, 1.570796, 1.668231],accel_mss,speed_ms,0,blend_radius_m)
    |   movel([0.097301, -1.385436, -2.571108, -0.755845, 1.570796, 1.668098],accel_mss,speed_ms,0,blend_radius_m)
    |   movel([0.097178, -1.385846, -2.570816, -0.755727, 1.570796, 1.667974],accel_mss,speed_ms,0,blend_radius_m)
    |   movel([0.097039, -1.386263, -2.570519, -0.755607, 1.570796, 1.667835],accel_mss,speed_ms,0,blend_radius_m)
    |   movel([0.096697, -1.387199, -2.569851, -0.755339, 1.570796, 1.667493],accel_mss,speed_ms,0,blend_radius_m)
    |   movel([0.096287, -1.388225, -2.569117, -0.755047, 1.570796, 1.667084],accel_mss,speed_ms,0,blend_radius_m)
    |   movel([0.095880, -1.389193, -2.568423, -0.754773, 1.570796, 1.666677],accel_mss,speed_ms,0,blend_radius_m)
    |   movel([0.095733, -1.389415, -2.568264, -0.754710, 1.570796, 1.666529],accel_mss,speed_ms,0,blend_radius_m)
    |   movel([0.095575, -1.389277, -2.568363, -0.754749, 1.570796, 1.666371],accel_mss,speed_ms,0,blend_radius_m)
    |   movel([0.095465, -1.388970, -2.568583, -0.754836, 1.570796, 1.666261],accel_mss,speed_ms,0,blend_radius_m)
    |   movel([0.095361, -1.388818, -2.568692, -0.754879, 1.570796, 1.666157],accel_mss,speed_ms,0,blend_radius_m)
    |   movel([0.095087, -1.388615, -2.568837, -0.754936, 1.570796, 1.665884],accel_mss,speed_ms,0,blend_radius_m)
    |   movel([0.094829, -1.388466, -2.568945, -0.754979, 1.570796, 1.665625],accel_mss,speed_ms,0,blend_radius_m)
    |   movel([0.094690, -1.388289, -2.569071, -0.755029, 1.570796, 1.665486],accel_mss,speed_ms,0,blend_radius_m)
    |   movel([0.094486, -1.387992, -2.569284, -0.755113, 1.570796, 1.665282],accel_mss,speed_ms,0,blend_radius_m)
    |   movel([0.093913, -1.387612, -2.569556, -0.755221, 1.570796, 1.664709],accel_mss,speed_ms,0,blend_radius_m)
    |   movel([0.093257, -1.387278, -2.569794, -0.755317, 1.570796, 1.664053],accel_mss,speed_ms,0,blend_radius_m)
    |   movel([0.092692, -1.387118, -2.569909, -0.755362, 1.570796, 1.663488],accel_mss,speed_ms,0,blend_radius_m)
    |   movel([0.092049, -1.387053, -2.569955, -0.755381, 1.570796, 1.662845],accel_mss,speed_ms,0,blend_radius_m)
    |   movel([0.091353, -1.387058, -2.569952, -0.755379, 1.570796, 1.662149],accel_mss,speed_ms,0,blend_radius_m)
    |   movel([0.090674, -1.387122, -2.569906, -0.755361, 1.570796, 1.661470],accel_mss,speed_ms,0,blend_radius_m)
    |   movel([0.090083, -1.387249, -2.569815, -0.755325, 1.570796, 1.660879],accel_mss,speed_ms,0,blend_radius_m)
    |   movel([0.089683, -1.387330, -2.569757, -0.755302, 1.570796, 1.660479],accel_mss,speed_ms,0,blend_radius_m)
    |   movel([0.089967, -1.387019, -2.569980, -0.755391, 1.570796, 1.660763],accel_mss,speed_ms,0,blend_radius_m)
    |   movel([0.090498, -1.386824, -2.570119, -0.755446, 1.570796, 1.661294],accel_mss,speed_ms,0,blend_radius_m)
    |   movel([0.091427, -1.386517, -2.570338, -0.755534, 1.570796, 1.662224],accel_mss,speed_ms,0,blend_radius_m)
    |   movel([0.093010, -1.385988, -2.570715, -0.755686, 1.570796, 1.663806],accel_mss,speed_ms,0,blend_radius_m)
    |   movel([0.094776, -1.385364, -2.571160, -0.755866, 1.570796, 1.665572],accel_mss,speed_ms,0,blend_radius_m)
    |   speed_ms = 0.003
    |   movel([0.094776, -1.372344, -2.565176, -0.774868, 1.570796, 1.665572],accel_mss,speed_ms,0,blend_radius_m)
    |   speed_ms = 1.000
    |   movel([0.094776, -1.347374, -2.552816, -0.812199, 1.570796, 1.665572],accel_mss,speed_ms,0,blend_radius_m)
    |   movel([0.095070, -1.346731, -2.553248, -0.812409, 1.570796, 1.665866],accel_mss,speed_ms,0,blend_radius_m)
    |   movel([0.095070, -1.371713, -2.565617, -0.775059, 1.570796, 1.665866],accel_mss,speed_ms,0,blend_radius_m)
    |   speed_ms = 0.003
    |   movel([0.095070, -1.381449, -2.570120, -0.760820, 1.570796, 1.665866],accel_mss,speed_ms,0,blend_radius_m)
    |   speed_ms = 0.007
    |   movel([0.096152, -1.381011, -2.570430, -0.760949, 1.570796, 1.666948],accel_mss,speed_ms,0,blend_radius_m)
    |   movel([0.097416, -1.380470, -2.570812, -0.761108, 1.570796, 1.668212],accel_mss,speed_ms,0,blend_radius_m)
    |   movel([0.097749, -1.380346, -2.570899, -0.761144, 1.570796, 1.668546],accel_mss,speed_ms,0,blend_radius_m)
    |   movel([0.098110, -1.380392, -2.570867, -0.761131, 1.570796, 1.668906],accel_mss,speed_ms,0,blend_radius_m)
    |   movel([0.098230, -1.380590, -2.570727, -0.761072, 1.570796, 1.669026],accel_mss,speed_ms,0,blend_radius_m)
    |   movel([0.098219, -1.380960, -2.570466, -0.760964, 1.570796, 1.669016],accel_mss,speed_ms,0,blend_radius_m)
    |   movel([0.098079, -1.381576, -2.570030, -0.760783, 1.570796, 1.668875],accel_mss,speed_ms,0,blend_radius_m)
    |   movel([0.097743, -1.382661, -2.569262, -0.760467, 1.570796, 1.668540],accel_mss,speed_ms,0,blend_radius_m)
    |   movel([0.097071, -1.384490, -2.567962, -0.759937, 1.570796, 1.667867],accel_mss,speed_ms,0,blend_radius_m)
    |   movel([0.096148, -1.386582, -2.566470, -0.759337, 1.570796, 1.666944],accel_mss,speed_ms,0,blend_radius_m)
    |   movel([0.095198, -1.388510, -2.565090, -0.758790, 1.570796, 1.665994],accel_mss,speed_ms,0,blend_radius_m)
    |   movel([0.094651, -1.389228, -2.564574, -0.758587, 1.570796, 1.665447],accel_mss,speed_ms,0,blend_radius_m)
    |   movel([0.094291, -1.389485, -2.564389, -0.758515, 1.570796, 1.665088],accel_mss,speed_ms,0,blend_radius_m)
    |   movel([0.093555, -1.389857, -2.564122, -0.758410, 1.570796, 1.664352],accel_mss,speed_ms,0,blend_radius_m)
    |   movel([0.092679, -1.390248, -2.563840, -0.758301, 1.570796, 1.663475],accel_mss,speed_ms,0,blend_radius_m)
    |   movel([0.091771, -1.390598, -2.563588, -0.758203, 1.570796, 1.662567],accel_mss,speed_ms,0,blend_radius_m)
    |   movel([0.091344, -1.390760, -2.563472, -0.758158, 1.570796, 1.662140],accel_mss,speed_ms,0,blend_radius_m)
    |   movel([0.091077, -1.390880, -2.563385, -0.758124, 1.570796, 1.661873],accel_mss,speed_ms,0,blend_radius_m)
    |   movel([0.090865, -1.391070, -2.563248, -0.758071, 1.570796, 1.661661],accel_mss,speed_ms,0,blend_radius_m)
    |   movel([0.091295, -1.391060, -2.563255, -0.758074, 1.570796, 1.662091],accel_mss,speed_ms,0,blend_radius_m)
    |   movel([0.091815, -1.390883, -2.563383, -0.758123, 1.570796, 1.662611],accel_mss,speed_ms,0,blend_radius_m)
    |   movel([0.092251, -1.390721, -2.563500, -0.758169, 1.570796, 1.663048],accel_mss,speed_ms,0,blend_radius_m)
    |   movel([0.092769, -1.390519, -2.563645, -0.758225, 1.570796, 1.663566],accel_mss,speed_ms,0,blend_radius_m)
    |   movel([0.093283, -1.390311, -2.563795, -0.758283, 1.570796, 1.664079],accel_mss,speed_ms,0,blend_radius_m)
    |   movel([0.093711, -1.390127, -2.563927, -0.758335, 1.570796, 1.664507],accel_mss,speed_ms,0,blend_radius_m)
    |   movel([0.094299, -1.389872, -2.564111, -0.758406, 1.570796, 1.665096],accel_mss,speed_ms,0,blend_radius_m)
    |   movel([0.094706, -1.389789, -2.564171, -0.758429, 1.570796, 1.665503],accel_mss,speed_ms,0,blend_radius_m)
    |   movel([0.094972, -1.389962, -2.564046, -0.758381, 1.570796, 1.665769],accel_mss,speed_ms,0,blend_radius_m)
    |   movel([0.095076, -1.390324, -2.563786, -0.758280, 1.570796, 1.665873],accel_mss,speed_ms,0,blend_radius_m)
    |   movel([0.095081, -1.390609, -2.563580, -0.758200, 1.570796, 1.665877],accel_mss,speed_ms,0,blend_radius_m)
    |   movel([0.095059, -1.390956, -2.563330, -0.758103, 1.570796, 1.665855],accel_mss,speed_ms,0,blend_radius_m)
    |   movel([0.094920, -1.391327, -2.563063, -0.758000, 1.570796, 1.665716],accel_mss,speed_ms,0,blend_radius_m)
    |   movel([0.093941, -1.392067, -2.562528, -0.757794, 1.570796, 1.664738],accel_mss,speed_ms,0,blend_radius_m)
    |   movel([0.092368, -1.392707, -2.562066, -0.757617, 1.570796, 1.663164],accel_mss,speed_ms,0,blend_radius_m)
    |   movel([0.090193, -1.393424, -2.561546, -0.757419, 1.570796, 1.660989],accel_mss,speed_ms,0,blend_radius_m)
    |   movel([0.087277, -1.394246, -2.560950, -0.757193, 1.570796, 1.658074],accel_mss,speed_ms,0,blend_radius_m)
    |   movel([0.085160, -1.394791, -2.560554, -0.757044, 1.570796, 1.655956],accel_mss,speed_ms,0,blend_radius_m)
    |   movel([0.083595, -1.395139, -2.560301, -0.756949, 1.570796, 1.654391],accel_mss,speed_ms,0,blend_radius_m)
    |   movel([0.082460, -1.395328, -2.560164, -0.756897, 1.570796, 1.653257],accel_mss,speed_ms,0,blend_radius_m)
    |   movel([0.081822, -1.395320, -2.560169, -0.756899, 1.570796, 1.652619],accel_mss,speed_ms,0,blend_radius_m)
    |   movel([0.081641, -1.395219, -2.560243, -0.756927, 1.570796, 1.652437],accel_mss,speed_ms,0,blend_radius_m)
    |   movel([0.081532, -1.395035, -2.560377, -0.756977, 1.570796, 1.652328],accel_mss,speed_ms,0,blend_radius_m)
    |   movel([0.081519, -1.394687, -2.560630, -0.757072, 1.570796, 1.652316],accel_mss,speed_ms,0,blend_radius_m)
    |   movel([0.081608, -1.394239, -2.560955, -0.757195, 1.570796, 1.652404],accel_mss,speed_ms,0,blend_radius_m)
    |   movel([0.081764, -1.393806, -2.561269, -0.757314, 1.570796, 1.652560],accel_mss,speed_ms,0,blend_radius_m)
    |   movel([0.081959, -1.393518, -2.561478, -0.757393, 1.570796, 1.652756],accel_mss,speed_ms,0,blend_radius_m)
    |   movel([0.082312, -1.393264, -2.561662, -0.757463, 1.570796, 1.653108],accel_mss,speed_ms,0,blend_radius_m)
    |   movel([0.082560, -1.393207, -2.561703, -0.757479, 1.570796, 1.653356],accel_mss,speed_ms,0,blend_radius_m)
    |   movel([0.083142, -1.393136, -2.561755, -0.757498, 1.570796, 1.653938],accel_mss,speed_ms,0,blend_radius_m)
    |   movel([0.083870, -1.393046, -2.561820, -0.757523, 1.570796, 1.654666],accel_mss,speed_ms,0,blend_radius_m)
    |   movel([0.084273, -1.392965, -2.561878, -0.757545, 1.570796, 1.655069],accel_mss,speed_ms,0,blend_radius_m)
    |   movel([0.084581, -1.392758, -2.562029, -0.757603, 1.570796, 1.655377],accel_mss,speed_ms,0,blend_radius_m)
    |   movel([0.084311, -1.392695, -2.562074, -0.757620, 1.570796, 1.655108],accel_mss,speed_ms,0,blend_radius_m)
    |   movel([0.083989, -1.392708, -2.562065, -0.757616, 1.570796, 1.654785],accel_mss,speed_ms,0,blend_radius_m)
    |   movel([0.083558, -1.392751, -2.562033, -0.757604, 1.570796, 1.654354],accel_mss,speed_ms,0,blend_radius_m)
    |   movel([0.083144, -1.392794, -2.562002, -0.757593, 1.570796, 1.653940],accel_mss,speed_ms,0,blend_radius_m)
    |   movel([0.082748, -1.392818, -2.561985, -0.757586, 1.570796, 1.653545],accel_mss,speed_ms,0,blend_radius_m)
    |   movel([0.082417, -1.392823, -2.561981, -0.757585, 1.570796, 1.653213],accel_mss,speed_ms,0,blend_radius_m)
    |   movel([0.081839, -1.392468, -2.562239, -0.757683, 1.570796, 1.652636],accel_mss,speed_ms,0,blend_radius_m)
    |   movel([0.081234, -1.391081, -2.563240, -0.758068, 1.570796, 1.652030],accel_mss,speed_ms,0,blend_radius_m)
    |   movel([0.080689, -1.389524, -2.564361, -0.758504, 1.570796, 1.651485],accel_mss,speed_ms,0,blend_radius_m)
    |   movel([0.080352, -1.388078, -2.565399, -0.758912, 1.570796, 1.651148],accel_mss,speed_ms,0,blend_radius_m)
    |   movel([0.080191, -1.386915, -2.566232, -0.759242, 1.570796, 1.650987],accel_mss,speed_ms,0,blend_radius_m)
    |   movel([0.080184, -1.386139, -2.566786, -0.759463, 1.570796, 1.650980],accel_mss,speed_ms,0,blend_radius_m)
    |   movel([0.080307, -1.385620, -2.567157, -0.759612, 1.570796, 1.651104],accel_mss,speed_ms,0,blend_radius_m)
    |   movel([0.080582, -1.385323, -2.567369, -0.759697, 1.570796, 1.651378],accel_mss,speed_ms,0,blend_radius_m)
    |   movel([0.081195, -1.385168, -2.567479, -0.759742, 1.570796, 1.651991],accel_mss,speed_ms,0,blend_radius_m)
    |   movel([0.081739, -1.385071, -2.567548, -0.759770, 1.570796, 1.652535],accel_mss,speed_ms,0,blend_radius_m)
    |   movel([0.082338, -1.384981, -2.567612, -0.759795, 1.570796, 1.653134],accel_mss,speed_ms,0,blend_radius_m)
    |   movel([0.083396, -1.384803, -2.567739, -0.759847, 1.570796, 1.654192],accel_mss,speed_ms,0,blend_radius_m)
    |   movel([0.084436, -1.384567, -2.567907, -0.759915, 1.570796, 1.655232],accel_mss,speed_ms,0,blend_radius_m)
    |   movel([0.085955, -1.384156, -2.568200, -0.760033, 1.570796, 1.656751],accel_mss,speed_ms,0,blend_radius_m)
    |   movel([0.089220, -1.383220, -2.568865, -0.760304, 1.570796, 1.660017],accel_mss,speed_ms,0,blend_radius_m)
    |   movel([0.092482, -1.382280, -2.569531, -0.760578, 1.570796, 1.663278],accel_mss,speed_ms,0,blend_radius_m)
    |   movel([0.094013, -1.381815, -2.569861, -0.760713, 1.570796, 1.664810],accel_mss,speed_ms,0,blend_radius_m)
    |   movel([0.095070, -1.381449, -2.570120, -0.760820, 1.570796, 1.665866],accel_mss,speed_ms,0,blend_radius_m)
    |   speed_ms = 0.003
    |   movel([0.095070, -1.384739, -2.571604, -0.756046, 1.570796, 1.665866],accel_mss,speed_ms,0,blend_radius_m)
    |   speed_ms = 0.007
    |   movel([0.096152, -1.384302, -2.571915, -0.756172, 1.570796, 1.666948],accel_mss,speed_ms,0,blend_radius_m)
    |   movel([0.097416, -1.383762, -2.572298, -0.756329, 1.570796, 1.668212],accel_mss,speed_ms,0,blend_radius_m)
    |   movel([0.097749, -1.383640, -2.572385, -0.756365, 1.570796, 1.668546],accel_mss,speed_ms,0,blend_radius_m)
    |   movel([0.098110, -1.383685, -2.572353, -0.756352, 1.570796, 1.668906],accel_mss,speed_ms,0,blend_radius_m)
    |   movel([0.098230, -1.383883, -2.572212, -0.756294, 1.570796, 1.669026],accel_mss,speed_ms,0,blend_radius_m)
    |   movel([0.098219, -1.384251, -2.571951, -0.756187, 1.570796, 1.669016],accel_mss,speed_ms,0,blend_radius_m)
    |   movel([0.098079, -1.384866, -2.571514, -0.756009, 1.570796, 1.668875],accel_mss,speed_ms,0,blend_radius_m)
    |   movel([0.097743, -1.385947, -2.570744, -0.755698, 1.570796, 1.668540],accel_mss,speed_ms,0,blend_radius_m)
    |   movel([0.097071, -1.387772, -2.569442, -0.755176, 1.570796, 1.667867],accel_mss,speed_ms,0,blend_radius_m)
    |   movel([0.096148, -1.389858, -2.567946, -0.754585, 1.570796, 1.666944],accel_mss,speed_ms,0,blend_radius_m)
    |   movel([0.095198, -1.391781, -2.566562, -0.754046, 1.570796, 1.665994],accel_mss,speed_ms,0,blend_radius_m)
    |   movel([0.094651, -1.392496, -2.566046, -0.753847, 1.570796, 1.665447],accel_mss,speed_ms,0,blend_radius_m)
    |   movel([0.094291, -1.392753, -2.565860, -0.753775, 1.570796, 1.665088],accel_mss,speed_ms,0,blend_radius_m)
    |   movel([0.093555, -1.393124, -2.565592, -0.753673, 1.570796, 1.664352],accel_mss,speed_ms,0,blend_radius_m)
    |   movel([0.092679, -1.393514, -2.565310, -0.753565, 1.570796, 1.663475],accel_mss,speed_ms,0,blend_radius_m)
    |   movel([0.091771, -1.393863, -2.565057, -0.753469, 1.570796, 1.662567],accel_mss,speed_ms,0,blend_radius_m)
    |   movel([0.091344, -1.394024, -2.564941, -0.753424, 1.570796, 1.662140],accel_mss,speed_ms,0,blend_radius_m)
    |   movel([0.091077, -1.394144, -2.564854, -0.753391, 1.570796, 1.661873],accel_mss,speed_ms,0,blend_radius_m)
    |   movel([0.090865, -1.394334, -2.564717, -0.753339, 1.570796, 1.661661],accel_mss,speed_ms,0,blend_radius_m)
    |   movel([0.091295, -1.394324, -2.564724, -0.753342, 1.570796, 1.662091],accel_mss,speed_ms,0,blend_radius_m)
    |   movel([0.091815, -1.394147, -2.564852, -0.753390, 1.570796, 1.662611],accel_mss,speed_ms,0,blend_radius_m)
    |   movel([0.092251, -1.393985, -2.564969, -0.753435, 1.570796, 1.663048],accel_mss,speed_ms,0,blend_radius_m)
    |   movel([0.092769, -1.393785, -2.565114, -0.753490, 1.570796, 1.663566],accel_mss,speed_ms,0,blend_radius_m)
    |   movel([0.093283, -1.393577, -2.565264, -0.753547, 1.570796, 1.664079],accel_mss,speed_ms,0,blend_radius_m)
    |   movel([0.093711, -1.393394, -2.565397, -0.753598, 1.570796, 1.664507],accel_mss,speed_ms,0,blend_radius_m)
    |   movel([0.094299, -1.393139, -2.565582, -0.753669, 1.570796, 1.665096],accel_mss,speed_ms,0,blend_radius_m)
    |   movel([0.094706, -1.393056, -2.565641, -0.753692, 1.570796, 1.665503],accel_mss,speed_ms,0,blend_radius_m)
    |   movel([0.094972, -1.393229, -2.565516, -0.753644, 1.570796, 1.665769],accel_mss,speed_ms,0,blend_radius_m)
    |   movel([0.095076, -1.393589, -2.565255, -0.753544, 1.570796, 1.665873],accel_mss,speed_ms,0,blend_radius_m)
    |   movel([0.095081, -1.393874, -2.565049, -0.753465, 1.570796, 1.665877],accel_mss,speed_ms,0,blend_radius_m)
    |   movel([0.095059, -1.394220, -2.564799, -0.753370, 1.570796, 1.665855],accel_mss,speed_ms,0,blend_radius_m)
    |   movel([0.094920, -1.394590, -2.564531, -0.753268, 1.570796, 1.665716],accel_mss,speed_ms,0,blend_radius_m)
    |   movel([0.093941, -1.395328, -2.563995, -0.753066, 1.570796, 1.664738],accel_mss,speed_ms,0,blend_radius_m)
    |   movel([0.092368, -1.395966, -2.563531, -0.752892, 1.570796, 1.663164],accel_mss,speed_ms,0,blend_radius_m)
    |   movel([0.090193, -1.396682, -2.563010, -0.752697, 1.570796, 1.660989],accel_mss,speed_ms,0,blend_radius_m)
    |   movel([0.087277, -1.397501, -2.562413, -0.752475, 1.570796, 1.658074],accel_mss,speed_ms,0,blend_radius_m)
    |   movel([0.085160, -1.398044, -2.562017, -0.752328, 1.570796, 1.655956],accel_mss,speed_ms,0,blend_radius_m)
    |   movel([0.083595, -1.398392, -2.561763, -0.752234, 1.570796, 1.654391],accel_mss,speed_ms,0,blend_radius_m)
    |   movel([0.082460, -1.398579, -2.561626, -0.752184, 1.570796, 1.653257],accel_mss,speed_ms,0,blend_radius_m)
    |   movel([0.081822, -1.398572, -2.561631, -0.752186, 1.570796, 1.652619],accel_mss,speed_ms,0,blend_radius_m)
    |   movel([0.081641, -1.398471, -2.561705, -0.752213, 1.570796, 1.652437],accel_mss,speed_ms,0,blend_radius_m)
    |   movel([0.081532, -1.398288, -2.561839, -0.752262, 1.570796, 1.652328],accel_mss,speed_ms,0,blend_radius_m)
    |   movel([0.081519, -1.397940, -2.562093, -0.752356, 1.570796, 1.652316],accel_mss,speed_ms,0,blend_radius_m)
    |   movel([0.081608, -1.397494, -2.562419, -0.752477, 1.570796, 1.652404],accel_mss,speed_ms,0,blend_radius_m)
    |   movel([0.081764, -1.397062, -2.562733, -0.752594, 1.570796, 1.652560],accel_mss,speed_ms,0,blend_radius_m)
    |   movel([0.081959, -1.396775, -2.562943, -0.752672, 1.570796, 1.652756],accel_mss,speed_ms,0,blend_radius_m)
    |   movel([0.082312, -1.396522, -2.563127, -0.752740, 1.570796, 1.653108],accel_mss,speed_ms,0,blend_radius_m)
    |   movel([0.082560, -1.396465, -2.563168, -0.752756, 1.570796, 1.653356],accel_mss,speed_ms,0,blend_radius_m)
    |   movel([0.083142, -1.396394, -2.563220, -0.752775, 1.570796, 1.653938],accel_mss,speed_ms,0,blend_radius_m)
    |   movel([0.083870, -1.396304, -2.563285, -0.752799, 1.570796, 1.654666],accel_mss,speed_ms,0,blend_radius_m)
    |   movel([0.084273, -1.396224, -2.563344, -0.752821, 1.570796, 1.655069],accel_mss,speed_ms,0,blend_radius_m)
    |   movel([0.084581, -1.396017, -2.563494, -0.752878, 1.570796, 1.655377],accel_mss,speed_ms,0,blend_radius_m)
    |   movel([0.084311, -1.395955, -2.563540, -0.752895, 1.570796, 1.655108],accel_mss,speed_ms,0,blend_radius_m)
    |   movel([0.083989, -1.395967, -2.563531, -0.752891, 1.570796, 1.654785],accel_mss,speed_ms,0,blend_radius_m)
    |   movel([0.083558, -1.396010, -2.563499, -0.752880, 1.570796, 1.654354],accel_mss,speed_ms,0,blend_radius_m)
    |   movel([0.083144, -1.396053, -2.563468, -0.752868, 1.570796, 1.653940],accel_mss,speed_ms,0,blend_radius_m)
    |   movel([0.082748, -1.396077, -2.563451, -0.752862, 1.570796, 1.653545],accel_mss,speed_ms,0,blend_radius_m)
    |   movel([0.082417, -1.396082, -2.563447, -0.752860, 1.570796, 1.653213],accel_mss,speed_ms,0,blend_radius_m)
    |   movel([0.081839, -1.395727, -2.563705, -0.752957, 1.570796, 1.652636],accel_mss,speed_ms,0,blend_radius_m)
    |   movel([0.081234, -1.394344, -2.564709, -0.753336, 1.570796, 1.652030],accel_mss,speed_ms,0,blend_radius_m)
    |   movel([0.080689, -1.392792, -2.565832, -0.753765, 1.570796, 1.651485],accel_mss,speed_ms,0,blend_radius_m)
    |   movel([0.080352, -1.391350, -2.566872, -0.754166, 1.570796, 1.651148],accel_mss,speed_ms,0,blend_radius_m)
    |   movel([0.080191, -1.390190, -2.567708, -0.754492, 1.570796, 1.650987],accel_mss,speed_ms,0,blend_radius_m)
    |   movel([0.080184, -1.389417, -2.568263, -0.754709, 1.570796, 1.650980],accel_mss,speed_ms,0,blend_radius_m)
    |   movel([0.080307, -1.388898, -2.568635, -0.754856, 1.570796, 1.651104],accel_mss,speed_ms,0,blend_radius_m)
    |   movel([0.080582, -1.388603, -2.568847, -0.754940, 1.570796, 1.651378],accel_mss,speed_ms,0,blend_radius_m)
    |   movel([0.081195, -1.388448, -2.568957, -0.754984, 1.570796, 1.651991],accel_mss,speed_ms,0,blend_radius_m)
    |   movel([0.081739, -1.388352, -2.569026, -0.755011, 1.570796, 1.652535],accel_mss,speed_ms,0,blend_radius_m)
    |   movel([0.082338, -1.388262, -2.569091, -0.755036, 1.570796, 1.653134],accel_mss,speed_ms,0,blend_radius_m)
    |   movel([0.083396, -1.388084, -2.569218, -0.755087, 1.570796, 1.654192],accel_mss,speed_ms,0,blend_radius_m)
    |   movel([0.084436, -1.387849, -2.569386, -0.755154, 1.570796, 1.655232],accel_mss,speed_ms,0,blend_radius_m)
    |   movel([0.085955, -1.387438, -2.569680, -0.755271, 1.570796, 1.656751],accel_mss,speed_ms,0,blend_radius_m)
    |   movel([0.089220, -1.386505, -2.570346, -0.755538, 1.570796, 1.660017],accel_mss,speed_ms,0,blend_radius_m)
    |   movel([0.092482, -1.385568, -2.571014, -0.755807, 1.570796, 1.663278],accel_mss,speed_ms,0,blend_radius_m)
    |   movel([0.094013, -1.385104, -2.571344, -0.755940, 1.570796, 1.664810],accel_mss,speed_ms,0,blend_radius_m)
    |   movel([0.095070, -1.384739, -2.571604, -0.756046, 1.570796, 1.665866],accel_mss,speed_ms,0,blend_radius_m)
    |   speed_ms = 0.003
    |   movel([0.095070, -1.371713, -2.565617, -0.775059, 1.570796, 1.665866],accel_mss,speed_ms,0,blend_radius_m)
    |   speed_ms = 1.000
    |   movel([0.095070, -1.346731, -2.553248, -0.812409, 1.570796, 1.665866],accel_mss,speed_ms,0,blend_radius_m)
    |   movel([0.089293, -1.355826, -2.547083, -0.809480, 1.570796, 1.660089],accel_mss,speed_ms,0,blend_radius_m)
    |   movel([0.089293, -1.380644, -2.559336, -0.772409, 1.570796, 1.660089],accel_mss,speed_ms,0,blend_radius_m)
    |   speed_ms = 0.003
    |   movel([0.089293, -1.390310, -2.563795, -0.758283, 1.570796, 1.660089],accel_mss,speed_ms,0,blend_radius_m)
    |   speed_ms = 0.007
    |   movel([0.089533, -1.390446, -2.563697, -0.758245, 1.570796, 1.660329],accel_mss,speed_ms,0,blend_radius_m)
    |   movel([0.089491, -1.390735, -2.563490, -0.758165, 1.570796, 1.660287],accel_mss,speed_ms,0,blend_radius_m)
    |   movel([0.089053, -1.390950, -2.563335, -0.758105, 1.570796, 1.659850],accel_mss,speed_ms,0,blend_radius_m)
    |   movel([0.088549, -1.391115, -2.563215, -0.758058, 1.570796, 1.659346],accel_mss,speed_ms,0,blend_radius_m)
    |   movel([0.088022, -1.391275, -2.563100, -0.758014, 1.570796, 1.658818],accel_mss,speed_ms,0,blend_radius_m)
    |   movel([0.087755, -1.391333, -2.563058, -0.757998, 1.570796, 1.658551],accel_mss,speed_ms,0,blend_radius_m)
    |   movel([0.087527, -1.391260, -2.563111, -0.758018, 1.570796, 1.658324],accel_mss,speed_ms,0,blend_radius_m)
    |   movel([0.087836, -1.390747, -2.563481, -0.758161, 1.570796, 1.658633],accel_mss,speed_ms,0,blend_radius_m)
    |   movel([0.088216, -1.390466, -2.563683, -0.758240, 1.570796, 1.659012],accel_mss,speed_ms,0,blend_radius_m)
    |   movel([0.088598, -1.390297, -2.563805, -0.758287, 1.570796, 1.659394],accel_mss,speed_ms,0,blend_radius_m)
    |   movel([0.088951, -1.390251, -2.563838, -0.758300, 1.570796, 1.659747],accel_mss,speed_ms,0,blend_radius_m)
    |   movel([0.089293, -1.390310, -2.563795, -0.758283, 1.570796, 1.660089],accel_mss,speed_ms,0,blend_radius_m)
    |   speed_ms = 0.003
    |   movel([0.089293, -1.393576, -2.565265, -0.753548, 1.570796, 1.660089],accel_mss,speed_ms,0,blend_radius_m)
    |   speed_ms = 0.007
    |   movel([0.089533, -1.393712, -2.565167, -0.753510, 1.570796, 1.660329],accel_mss,speed_ms,0,blend_radius_m)
    |   movel([0.089491, -1.393999, -2.564959, -0.753431, 1.570796, 1.660287],accel_mss,speed_ms,0,blend_radius_m)
    |   movel([0.089053, -1.394214, -2.564804, -0.753372, 1.570796, 1.659850],accel_mss,speed_ms,0,blend_radius_m)
    |   movel([0.088549, -1.394379, -2.564684, -0.753326, 1.570796, 1.659346],accel_mss,speed_ms,0,blend_radius_m)
    |   movel([0.088022, -1.394539, -2.564568, -0.753283, 1.570796, 1.658818],accel_mss,speed_ms,0,blend_radius_m)
    |   movel([0.087755, -1.394596, -2.564526, -0.753267, 1.570796, 1.658551],accel_mss,speed_ms,0,blend_radius_m)
    |   movel([0.087527, -1.394523, -2.564579, -0.753287, 1.570796, 1.658324],accel_mss,speed_ms,0,blend_radius_m)
